LIN {X 0,Y 367.535,Z 523.641,A -85,B 0,C 180,E1 -12888.968,E2 -12888.968} C_VEL
LIN {X 0,Y 367.844,Z 521.457,A -85,B 0,C 180,E1 -12890.579,E2 -12890.579} C_VEL
LIN {X 0,Y 368.245,Z 517.815,A -85,B 0,C 180,E1 -12892.437,E2 -12892.437} C_VEL
LIN {X 0,Y 368.494,Z 515.813,A -85,B 0,C 180,E1 -12893.236,E2 -12893.236} C_VEL
LIN {X 0,Y 368.092,Z 513.552,A -85,B 0,C 180,E1 -12894.082,E2 -12894.082} C_VEL
LIN {X 0,Y 365.767,Z 509.524,A -85,B 0,C 180,E1 -12895.454,E2 -12895.454} C_VEL
LIN {X 0,Y 363.625,Z 504.962,A -85,B 0,C 180,E1 -12896.791,E2 -12896.791} C_VEL
LIN {X 0,Y 363.51,Z 501.685,A -85,B 0,C 180,E1 -12897.571,E2 -12897.571} C_VEL
LIN {X 0,Y 364.573,Z 493.787,A -85,B 0,C 180,E1 -12899.125,E2 -12899.125} C_VEL
LIN {X 0,Y 365.898,Z 483.754,A -85,B 0,C 180,E1 -12900.707,E2 -12900.707} C_VEL
LIN {X 0,Y 367.105,Z 474.13,A -85,B 0,C 180,E1 -12901.926,E2 -12901.926} C_VEL
LIN {X 0,Y 368.273,Z 463.742,A -85,B 0,C 180,E1 -12902.986,E2 -12902.986} C_VEL
LIN {X 0,Y 369.362,Z 451.282,A -85,B 0,C 180,E1 -12903.979,E2 -12903.979} C_VEL
LIN {X 0,Y 370.27,Z 438.997,A -85,B 0,C 180,E1 -12904.707,E2 -12904.707} C_VEL
LIN {X 0,Y 370.88,Z 426.339,A -85,B 0,C 180,E1 -12905.229,E2 -12905.229} C_VEL
LIN {X 0,Y 371.342,Z 411.465,A -85,B 0,C 180,E1 -12905.584,E2 -12905.584} C_VEL
LIN {X 0,Y 372.709,Z 340.608,A -85,B 0,C 180,E1 -12906.985,E2 -12906.985} C_VEL
LIN {X 0,Y 369.758,Z 328.428,A -85,B 0,C 180,E1 -12907.469,E2 -12907.469} C_VEL
LIN {X 0,Y 363.989,Z 314.826,A -85,B 0,C 180,E1 -12908.246,E2 -12908.246} C_VEL
LIN {X 0,Y 361.815,Z 305.413,A -85,B 0,C 180,E1 -12910.911,E2 -12910.911} C_VEL
LIN {X 0,Y 361.802,Z 305.418,A -85,B 0,C 180,E1 -12914.368,E2 -12914.368} C_VEL
LIN {X 0,Y 361.818,Z 305.416,A -85,B 0,C 180,E1 -12917.568,E2 -12917.568} C_VEL
LIN {X 0,Y 361.83,Z 305.417,A -85,B 0,C 180,E1 -12921.571,E2 -12921.571} C_VEL
LIN {X 0,Y 361.858,Z 305.393,A -85,B 0,C 180,E1 -12924.655,E2 -12924.655} C_VEL
LIN {X 0,Y 361.824,Z 305.409,A -85,B 0,C 180,E1 -12928.37,E2 -12928.37} C_VEL
LIN {X 0,Y 361.853,Z 305.409,A -85,B 0,C 180,E1 -12930.951,E2 -12930.951} C_VEL
LIN {X 0,Y 361.87,Z 305.403,A -85,B 0,C 180,E1 -12934.706,E2 -12934.706} C_VEL
LIN {X 0,Y 361.847,Z 305.405,A -85,B 0,C 180,E1 -12938.344,E2 -12938.344} C_VEL
LIN {X 0,Y 361.954,Z 305.397,A -85,B 0,C 180,E1 -12942.061,E2 -12942.061} C_VEL
LIN {X 0,Y 361.984,Z 305.396,A -85,B 0,C 180,E1 -12946.101,E2 -12946.101} C_VEL
LIN {X 0,Y 362.018,Z 305.389,A -85,B 0,C 180,E1 -12949.938,E2 -12949.938} C_VEL
LIN {X 0,Y 362.12,Z 305.366,A -85,B 0,C 180,E1 -12953.313,E2 -12953.313} C_VEL
LIN {X 0,Y 362.266,Z 305.351,A -85,B 0,C 180,E1 -12957.777,E2 -12957.777} C_VEL
LIN {X 0,Y 362.413,Z 305.337,A -85,B 0,C 180,E1 -12960,E2 -12960} C_VEL
LIN {X 0,Y 362.266,Z 305.355,A -85,B 0,C 180,E1 -12962.224,E2 -12962.224} C_VEL
LIN {X 0,Y 362.156,Z 305.371,A -85,B 0,C 180,E1 -12966.687,E2 -12966.687} C_VEL
LIN {X 0,Y 362.06,Z 305.376,A -85,B 0,C 180,E1 -12968.934,E2 -12968.934} C_VEL
LIN {X 0,Y 361.948,Z 305.397,A -85,B 0,C 180,E1 -12972.333,E2 -12972.333} C_VEL
LIN {X 0,Y 361.949,Z 305.39,A -85,B 0,C 180,E1 -12974.621,E2 -12974.621} C_VEL
LIN {X 0,Y 361.947,Z 305.392,A -85,B 0,C 180,E1 -12978.1,E2 -12978.1} C_VEL
LIN {X 0,Y 361.88,Z 305.405,A -85,B 0,C 180,E1 -12981.654,E2 -12981.654} C_VEL
LIN {X 0,Y 361.916,Z 305.404,A -85,B 0,C 180,E1 -12985.291,E2 -12985.291} C_VEL
LIN {X 0,Y 361.911,Z 305.394,A -85,B 0,C 180,E1 -12987.779,E2 -12987.779} C_VEL
LIN {X 0,Y 361.85,Z 305.405,A -85,B 0,C 180,E1 -12991.629,E2 -12991.629} C_VEL
LIN {X 0,Y 361.865,Z 305.408,A -85,B 0,C 180,E1 -12995.346,E2 -12995.346} C_VEL
LIN {X 0,Y 361.866,Z 305.409,A -85,B 0,C 180,E1 -12999.029,E2 -12999.029} C_VEL
LIN {X 0,Y 361.849,Z 305.408,A -85,B 0,C 180,E1 -13002.437,E2 -13002.437} C_VEL
LIN {X 0,Y 361.891,Z 305.393,A -85,B 0,C 180,E1 -13005.935,E2 -13005.935} C_VEL
LIN {X 0,Y 361.899,Z 305.401,A -85,B 0,C 180,E1 -13009.233,E2 -13009.233} C_VEL
LIN {X 0,Y 361.863,Z 305.407,A -85,B 0,C 180,E1 -13012.984,E2 -13012.984} C_VEL
LIN {X 0,Y 361.853,Z 305.407,A -85,B 0,C 180,E1 -13016.633,E2 -13016.633} C_VEL
LIN {X 0,Y 361.904,Z 305.519,A -85,B 0,C 180,E1 -13018.541,E2 -13018.541} C_VEL
LIN {X 0,Y 364.797,Z 317.675,A -85,B 0,C 180,E1 -13021.838,E2 -13021.838} C_VEL
LIN {X 0,Y 366.633,Z 327.228,A -85,B 0,C 180,E1 -13024.283,E2 -13024.283} C_VEL
LIN {X 0,Y 366.075,Z 334.395,A -85,B 0,C 180,E1 -13025.925,E2 -13025.925} C_VEL
LIN {X 0,Y 365.502,Z 339.003,A -85,B 0,C 180,E1 -13026.956,E2 -13026.956} C_VEL
LIN {X 0,Y 369.726,Z 359.775,A -85,B 0,C 180,E1 -13027.733,E2 -13027.733} C_VEL
LIN {X 0,Y 372.145,Z 375.173,A -85,B 0,C 180,E1 -13028.239,E2 -13028.239} C_VEL
LIN {X 0,Y 370.626,Z 447.548,A -85,B 0,C 180,E1 -13029.683,E2 -13029.683} C_VEL
LIN {X 0,Y 369.963,Z 460.734,A -85,B 0,C 180,E1 -13030.152,E2 -13030.152} C_VEL
LIN {X 0,Y 368.926,Z 473.426,A -85,B 0,C 180,E1 -13030.817,E2 -13030.817} C_VEL
LIN {X 0,Y 367.825,Z 484.734,A -85,B 0,C 180,E1 -13031.625,E2 -13031.625} C_VEL
LIN {X 0,Y 366.507,Z 496.397,A -85,B 0,C 180,E1 -13032.711,E2 -13032.711} C_VEL
LIN {X 0,Y 365.178,Z 506.891,A -85,B 0,C 180,E1 -13033.941,E2 -13033.941} C_VEL
LIN {X 0,Y 364.137,Z 515.532,A -85,B 0,C 180,E1 -13035.191,E2 -13035.191} C_VEL
LIN {X 0,Y 363.149,Z 523.447,A -85,B 0,C 180,E1 -13036.573,E2 -13036.573} C_VEL
LIN {X 0,Y 362.018,Z 531.267,A -85,B 0,C 180,E1 -13038.24,E2 -13038.24} C_VEL
LIN {X 0,Y 361.281,Z 537.541,A -85,B 0,C 180,E1 -13039.919,E2 -13039.919} C_VEL
LIN {X 0,Y 360.808,Z 542.555,A -85,B 0,C 180,E1 -13041.601,E2 -13041.601} C_VEL
LIN {X 0,Y 360.498,Z 546.453,A -85,B 0,C 180,E1 -13043.284,E2 -13043.284} C_VEL
LIN {X 0,Y 360.365,Z 550.078,A -85,B 0,C 180,E1 -13045.528,E2 -13045.528} C_VEL
LIN {X 0,Y 360.301,Z 551.276,A -85,B 0,C 180,E1 -13046.647,E2 -13046.647} C_VEL
LIN {X 0,Y 360.358,Z 552.408,A -85,B 0,C 180,E1 -13048.884,E2 -13048.884} C_VEL
LIN {X 0,Y 360.423,Z 552.394,A -85,B 0,C 180,E1 -13050.002,E2 -13050.002} C_VEL
LIN {X 0,Y 360.39,Z 551.986,A -85,B 0,C 180,E1 -13051.119,E2 -13051.119} C_VEL
LIN {X 0,Y 360.327,Z 551.136,A -85,B 0,C 180,E1 -13052.237,E2 -13052.237} C_VEL
LIN {X 0,Y 360.322,Z 549.88,A -85,B 0,C 180,E1 -13053.356,E2 -13053.356} C_VEL
LIN {X 0,Y 360.376,Z 547.203,A -85,B 0,C 180,E1 -13055.036,E2 -13055.036} C_VEL
LIN {X 0,Y 360.499,Z 543.49,A -85,B 0,C 180,E1 -13056.719,E2 -13056.719} C_VEL
LIN {X 0,Y 360.749,Z 538.639,A -85,B 0,C 180,E1 -13058.403,E2 -13058.403} C_VEL
LIN {X 0,Y 361.16,Z 532.502,A -85,B 0,C 180,E1 -13060.088,E2 -13060.088} C_VEL
LIN {X 0,Y 361.765,Z 524.858,A -85,B 0,C 180,E1 -13061.772,E2 -13061.772} C_VEL
LIN {X 0,Y 362.468,Z 517.035,A -85,B 0,C 180,E1 -13063.171,E2 -13063.171} C_VEL
LIN {X 0,Y 363.412,Z 507.472,A -85,B 0,C 180,E1 -13064.562,E2 -13064.562} C_VEL
LIN {X 0,Y 364.246,Z 496.828,A -85,B 0,C 180,E1 -13065.817,E2 -13065.817} C_VEL
LIN {X 0,Y 365.222,Z 484.96,A -85,B 0,C 180,E1 -13066.922,E2 -13066.922} C_VEL
LIN {X 0,Y 366.15,Z 472.226,A -85,B 0,C 180,E1 -13067.814,E2 -13067.814} C_VEL
LIN {X 0,Y 366.97,Z 459.529,A -85,B 0,C 180,E1 -13068.459,E2 -13068.459} C_VEL
LIN {X 0,Y 367.431,Z 447.489,A -85,B 0,C 180,E1 -13068.868,E2 -13068.868} C_VEL
LIN {X 0,Y 368.577,Z 374.068,A -85,B 0,C 180,E1 -13070.315,E2 -13070.315} C_VEL
LIN {X 0,Y 363.856,Z 339.626,A -85,B 0,C 180,E1 -13071.264,E2 -13071.264} C_VEL
LIN {X 0,Y 365.182,Z 323.829,A -85,B 0,C 180,E1 -13074.747,E2 -13074.747} C_VEL
LIN {X 0,Y 364.808,Z 319.729,A -85,B 0,C 180,E1 -13075.697,E2 -13075.697} C_VEL
LIN {X 0,Y 362.061,Z 305.992,A -85,B 0,C 180,E1 -13079.032,E2 -13079.032} C_VEL
LIN {X 0,Y 361.931,Z 305.4,A -85,B 0,C 180,E1 -13079.222,E2 -13079.222} C_VEL
LIN {X 0,Y 361.865,Z 305.405,A -85,B 0,C 180,E1 -13083.37,E2 -13083.37} C_VEL
LIN {X 0,Y 361.872,Z 305.405,A -85,B 0,C 180,E1 -13087.019,E2 -13087.019} C_VEL
LIN {X 0,Y 361.86,Z 305.407,A -85,B 0,C 180,E1 -13089.862,E2 -13089.862} C_VEL
LIN {X 0,Y 361.842,Z 305.412,A -85,B 0,C 180,E1 -13092.83,E2 -13092.83} C_VEL
LIN {X 0,Y 361.824,Z 305.411,A -85,B 0,C 180,E1 -13095.947,E2 -13095.947} C_VEL
LIN {X 0,Y 361.842,Z 305.41,A -85,B 0,C 180,E1 -13099.245,E2 -13099.245} C_VEL
LIN {X 0,Y 361.87,Z 305.411,A -85,B 0,C 180,E1 -13102.778,E2 -13102.778} C_VEL
LIN {X 0,Y 361.86,Z 305.406,A -85,B 0,C 180,E1 -13105.72,E2 -13105.72} C_VEL
LIN {X 0,Y 361.881,Z 305.405,A -85,B 0,C 180,E1 -13109.672,E2 -13109.672} C_VEL
LIN {X 0,Y 361.961,Z 305.398,A -85,B 0,C 180,E1 -13113.475,E2 -13113.475} C_VEL
LIN {X 0,Y 361.886,Z 305.407,A -85,B 0,C 180,E1 -13117.144,E2 -13117.144} C_VEL
LIN {X 0,Y 361.892,Z 305.402,A -85,B 0,C 180,E1 -13120.722,E2 -13120.722} C_VEL
LIN {X 0,Y 361.95,Z 305.396,A -85,B 0,C 180,E1 -13124.226,E2 -13124.226} C_VEL
LIN {X 0,Y 362.006,Z 305.388,A -85,B 0,C 180,E1 -13126.528,E2 -13126.528} C_VEL
LIN {X 0,Y 362.036,Z 305.389,A -85,B 0,C 180,E1 -13129.938,E2 -13129.938} C_VEL
LIN {X 0,Y 362.131,Z 305.373,A -85,B 0,C 180,E1 -13133.313,E2 -13133.313} C_VEL
LIN {X 0,Y 362.286,Z 305.357,A -85,B 0,C 180,E1 -13137.776,E2 -13137.776} C_VEL
LIN {X 0,Y 362.43,Z 305.341,A -85,B 0,C 180,E1 -13140,E2 -13140} C_VEL
LIN {X 0,Y 362.285,Z 305.36,A -85,B 0,C 180,E1 -13142.223,E2 -13142.223} C_VEL
LIN {X 0,Y 362.154,Z 305.372,A -85,B 0,C 180,E1 -13146.686,E2 -13146.686} C_VEL
LIN {X 0,Y 362.006,Z 305.391,A -85,B 0,C 180,E1 -13150.063,E2 -13150.063} C_VEL
LIN {X 0,Y 362.004,Z 305.389,A -85,B 0,C 180,E1 -13153.898,E2 -13153.898} C_VEL
LIN {X 0,Y 361.934,Z 305.401,A -85,B 0,C 180,E1 -13156.934,E2 -13156.934} C_VEL
LIN {X 0,Y 361.892,Z 305.405,A -85,B 0,C 180,E1 -13160.46,E2 -13160.46} C_VEL
LIN {X 0,Y 361.899,Z 305.401,A -85,B 0,C 180,E1 -13164.112,E2 -13164.112} C_VEL
LIN {X 0,Y 361.947,Z 305.399,A -85,B 0,C 180,E1 -13166.721,E2 -13166.721} C_VEL
LIN {X 0,Y 361.878,Z 305.404,A -85,B 0,C 180,E1 -13170.327,E2 -13170.327} C_VEL
LIN {X 0,Y 361.859,Z 305.406,A -85,B 0,C 180,E1 -13174.28,E2 -13174.28} C_VEL
LIN {X 0,Y 361.868,Z 305.411,A -85,B 0,C 180,E1 -13177.222,E2 -13177.222} C_VEL
LIN {X 0,Y 361.84,Z 305.409,A -85,B 0,C 180,E1 -13180.755,E2 -13180.755} C_VEL
LIN {X 0,Y 361.821,Z 305.411,A -85,B 0,C 180,E1 -13184.368,E2 -13184.368} C_VEL
LIN {X 0,Y 361.84,Z 305.414,A -85,B 0,C 180,E1 -13187.567,E2 -13187.567} C_VEL
LIN {X 0,Y 361.872,Z 305.405,A -85,B 0,C 180,E1 -13190.973,E2 -13190.973} C_VEL
LIN {X 0,Y 361.878,Z 305.404,A -85,B 0,C 180,E1 -13194.654,E2 -13194.654} C_VEL
LIN {X 0,Y 361.842,Z 305.411,A -85,B 0,C 180,E1 -13198.369,E2 -13198.369} C_VEL
LIN {X 0,Y 361.912,Z 305.406,A -85,B 0,C 180,E1 -13202.22,E2 -13202.22} C_VEL
LIN {X 0,Y 361.931,Z 305.399,A -85,B 0,C 180,E1 -13204.709,E2 -13204.709} C_VEL
LIN {X 0,Y 361.902,Z 305.408,A -85,B 0,C 180,E1 -13208.346,E2 -13208.346} C_VEL
LIN {X 0,Y 361.971,Z 305.395,A -85,B 0,C 180,E1 -13212.06,E2 -13212.06} C_VEL
LIN {X 0,Y 362,Z 305.39,A -85,B 0,C 180,E1 -13216.1,E2 -13216.1} C_VEL
LIN {X 0,Y 362.002,Z 305.389,A -85,B 0,C 180,E1 -13219.936,E2 -13219.936} C_VEL
LIN {X 0,Y 362.087,Z 305.512,A -85,B 0,C 180,E1 -13221.461,E2 -13221.461} C_VEL
LIN {X 0,Y 363.79,Z 314.739,A -85,B 0,C 180,E1 -13223.84,E2 -13223.84} C_VEL
LIN {X 0,Y 365.852,Z 322.952,A -85,B 0,C 180,E1 -13224.111,E2 -13224.111} C_VEL
LIN {X 0,Y 369.039,Z 340.026,A -85,B 0,C 180,E1 -13224.613,E2 -13224.613} C_VEL
LIN {X 0,Y 367.633,Z 422.051,A -85,B 0,C 180,E1 -13226.231,E2 -13226.231} C_VEL
LIN {X 0,Y 367.087,Z 435.227,A -85,B 0,C 180,E1 -13226.706,E2 -13226.706} C_VEL
LIN {X 0,Y 366.558,Z 447.799,A -85,B 0,C 180,E1 -13227.388,E2 -13227.388} C_VEL
LIN {X 0,Y 365.821,Z 459.62,A -85,B 0,C 180,E1 -13228.258,E2 -13228.258} C_VEL
LIN {X 0,Y 364.903,Z 470.713,A -85,B 0,C 180,E1 -13229.309,E2 -13229.309} C_VEL
LIN {X 0,Y 363.959,Z 481.189,A -85,B 0,C 180,E1 -13230.552,E2 -13230.552} C_VEL
LIN {X 0,Y 363.107,Z 490.613,A -85,B 0,C 180,E1 -13231.939,E2 -13231.939} C_VEL
LIN {X 0,Y 362.216,Z 499.705,A -85,B 0,C 180,E1 -13233.614,E2 -13233.614} C_VEL
LIN {X 0,Y 361.528,Z 507.037,A -85,B 0,C 180,E1 -13235.296,E2 -13235.296} C_VEL
LIN {X 0,Y 361.166,Z 513.125,A -85,B 0,C 180,E1 -13237.061,E2 -13237.061} C_VEL
LIN {X 0,Y 360.72,Z 518.155,A -85,B 0,C 180,E1 -13238.965,E2 -13238.965} C_VEL
LIN {X 0,Y 360.511,Z 520.505,A -85,B 0,C 180,E1 -13240.103,E2 -13240.103} C_VEL
LIN {X 0,Y 360.403,Z 522.413,A -85,B 0,C 180,E1 -13241.243,E2 -13241.243} C_VEL
LIN {X 0,Y 360.295,Z 524.217,A -85,B 0,C 180,E1 -13242.758,E2 -13242.758} C_VEL
LIN {X 0,Y 360.201,Z 525.48,A -85,B 0,C 180,E1 -13244.692,E2 -13244.692} C_VEL
LIN {X 0,Y 360.218,Z 525.667,A -85,B 0,C 180,E1 -13245.85,E2 -13245.85} C_VEL
LIN {X 0,Y 360.27,Z 525.382,A -85,B 0,C 180,E1 -13247.085,E2 -13247.085} C_VEL
LIN {X 0,Y 360.499,Z 523.665,A -85,B 0,C 180,E1 -13249.353,E2 -13249.353} C_VEL
LIN {X 0,Y 360.805,Z 521.693,A -85,B 0,C 180,E1 -13250.776,E2 -13250.776} C_VEL
LIN {X 0,Y 361.311,Z 517.534,A -85,B 0,C 180,E1 -13252.892,E2 -13252.892} C_VEL
LIN {X 0,Y 361.97,Z 512.677,A -85,B 0,C 180,E1 -13254.671,E2 -13254.671} C_VEL
LIN {X 0,Y 362.839,Z 506.421,A -85,B 0,C 180,E1 -13256.453,E2 -13256.453} C_VEL
LIN {X 0,Y 363.51,Z 501.685,A -85,B 0,C 180,E1 -13257.571,E2 -13257.571} C_VEL
LIN {X 0,Y 363.434,Z 498.283,A -85,B 0,C 180,E1 -13258.333,E2 -13258.333} C_VEL
LIN {X 0,Y 361.524,Z 492.515,A -85,B 0,C 180,E1 -13259.574,E2 -13259.574} C_VEL
LIN {X 0,Y 359.6,Z 486.162,A -85,B 0,C 180,E1 -13260.746,E2 -13260.746} C_VEL
LIN {X 0,Y 359.49,Z 481.841,A -85,B 0,C 180,E1 -13261.388,E2 -13261.388} C_VEL
LIN {X 0,Y 360.854,Z 470.901,A -85,B 0,C 180,E1 -13262.712,E2 -13262.712} C_VEL
LIN {X 0,Y 362.095,Z 459.975,A -85,B 0,C 180,E1 -13263.76,E2 -13263.76} C_VEL
LIN {X 0,Y 363.096,Z 448.05,A -85,B 0,C 180,E1 -13264.648,E2 -13264.648} C_VEL
LIN {X 0,Y 363.996,Z 435.03,A -85,B 0,C 180,E1 -13265.352,E2 -13265.352} C_VEL
LIN {X 0,Y 364.566,Z 422.079,A -85,B 0,C 180,E1 -13265.82,E2 -13265.82} C_VEL
LIN {X 0,Y 366.353,Z 341.95,A -85,B 0,C 180,E1 -13267.441,E2 -13267.441} C_VEL
LIN {X 0,Y 363.742,Z 331.236,A -85,B 0,C 180,E1 -13267.882,E2 -13267.882} C_VEL
LIN {X 0,Y 356.868,Z 315.147,A -85,B 0,C 180,E1 -13268.828,E2 -13268.828} C_VEL
LIN {X 0,Y 354.764,Z 306.292,A -85,B 0,C 180,E1 -13271.421,E2 -13271.421} C_VEL
LIN {X 0,Y 354.749,Z 306.296,A -85,B 0,C 180,E1 -13274.504,E2 -13274.504} C_VEL
LIN {X 0,Y 354.776,Z 306.295,A -85,B 0,C 180,E1 -13277.66,E2 -13277.66} C_VEL
LIN {X 0,Y 354.773,Z 306.293,A -85,B 0,C 180,E1 -13280.661,E2 -13280.661} C_VEL
LIN {X 0,Y 354.806,Z 306.271,A -85,B 0,C 180,E1 -13284.301,E2 -13284.301} C_VEL
LIN {X 0,Y 354.774,Z 306.294,A -85,B 0,C 180,E1 -13287.666,E2 -13287.666} C_VEL
LIN {X 0,Y 354.788,Z 306.288,A -85,B 0,C 180,E1 -13291.614,E2 -13291.614} C_VEL
LIN {X 0,Y 354.821,Z 306.281,A -85,B 0,C 180,E1 -13295.656,E2 -13295.656} C_VEL
LIN {X 0,Y 354.813,Z 306.279,A -85,B 0,C 180,E1 -13299.113,E2 -13299.113} C_VEL
LIN {X 0,Y 354.884,Z 306.271,A -85,B 0,C 180,E1 -13302.719,E2 -13302.719} C_VEL
LIN {X 0,Y 354.937,Z 306.272,A -85,B 0,C 180,E1 -13306.255,E2 -13306.255} C_VEL
LIN {X 0,Y 354.965,Z 306.266,A -85,B 0,C 180,E1 -13309.736,E2 -13309.736} C_VEL
LIN {X 0,Y 355.085,Z 306.242,A -85,B 0,C 180,E1 -13313.18,E2 -13313.18} C_VEL
LIN {X 0,Y 355.229,Z 306.227,A -85,B 0,C 180,E1 -13317.733,E2 -13317.733} C_VEL
LIN {X 0,Y 355.383,Z 306.212,A -85,B 0,C 180,E1 -13320,E2 -13320} C_VEL
LIN {X 0,Y 355.229,Z 306.23,A -85,B 0,C 180,E1 -13322.268,E2 -13322.268} C_VEL
LIN {X 0,Y 355.123,Z 306.246,A -85,B 0,C 180,E1 -13326.82,E2 -13326.82} C_VEL
LIN {X 0,Y 355.002,Z 306.255,A -85,B 0,C 180,E1 -13329.113,E2 -13329.113} C_VEL
LIN {X 0,Y 354.908,Z 306.271,A -85,B 0,C 180,E1 -13332.582,E2 -13332.582} C_VEL
LIN {X 0,Y 354.876,Z 306.278,A -85,B 0,C 180,E1 -13336.097,E2 -13336.097} C_VEL
LIN {X 0,Y 354.894,Z 306.27,A -85,B 0,C 180,E1 -13338.473,E2 -13338.473} C_VEL
LIN {X 0,Y 354.822,Z 306.284,A -85,B 0,C 180,E1 -13342.107,E2 -13342.107} C_VEL
LIN {X 0,Y 354.888,Z 306.277,A -85,B 0,C 180,E1 -13345.829,E2 -13345.829} C_VEL
LIN {X 0,Y 354.844,Z 306.285,A -85,B 0,C 180,E1 -13349.68,E2 -13349.68} C_VEL
LIN {X 0,Y 354.82,Z 306.29,A -85,B 0,C 180,E1 -13353.684,E2 -13353.684} C_VEL
LIN {X 0,Y 354.792,Z 306.288,A -85,B 0,C 180,E1 -13356.461,E2 -13356.461} C_VEL
LIN {X 0,Y 354.815,Z 306.287,A -85,B 0,C 180,E1 -13359.425,E2 -13359.425} C_VEL
LIN {X 0,Y 354.8,Z 306.287,A -85,B 0,C 180,E1 -13362.872,E2 -13362.872} C_VEL
LIN {X 0,Y 354.833,Z 306.272,A -85,B 0,C 180,E1 -13366.117,E2 -13366.117} C_VEL
LIN {X 0,Y 354.851,Z 306.279,A -85,B 0,C 180,E1 -13369.191,E2 -13369.191} C_VEL
LIN {X 0,Y 354.803,Z 306.29,A -85,B 0,C 180,E1 -13372.404,E2 -13372.404} C_VEL
LIN {X 0,Y 354.807,Z 306.292,A -85,B 0,C 180,E1 -13374.943,E2 -13374.943} C_VEL
LIN {X 0,Y 354.862,Z 306.413,A -85,B 0,C 180,E1 -13378.037,E2 -13378.037} C_VEL
LIN {X 0,Y 357.895,Z 319.073,A -85,B 0,C 180,E1 -13381.565,E2 -13381.565} C_VEL
LIN {X 0,Y 359.716,Z 328.332,A -85,B 0,C 180,E1 -13383.993,E2 -13383.993} C_VEL
LIN {X 0,Y 359.647,Z 331.913,A -85,B 0,C 180,E1 -13384.85,E2 -13384.85} C_VEL
LIN {X 0,Y 358.826,Z 338.677,A -85,B 0,C 180,E1 -13386.402,E2 -13386.402} C_VEL
LIN {X 0,Y 363.247,Z 360.149,A -85,B 0,C 180,E1 -13387.246,E2 -13387.246} C_VEL
LIN {X 0,Y 365.738,Z 376.161,A -85,B 0,C 180,E1 -13387.786,E2 -13387.786} C_VEL
LIN {X 0,Y 364.147,Z 447.404,A -85,B 0,C 180,E1 -13389.231,E2 -13389.231} C_VEL
LIN {X 0,Y 363.443,Z 460.548,A -85,B 0,C 180,E1 -13389.706,E2 -13389.706} C_VEL
LIN {X 0,Y 362.33,Z 473.223,A -85,B 0,C 180,E1 -13390.381,E2 -13390.381} C_VEL
LIN {X 0,Y 361.128,Z 485.309,A -85,B 0,C 180,E1 -13391.272,E2 -13391.272} C_VEL
LIN {X 0,Y 359.74,Z 496.806,A -85,B 0,C 180,E1 -13392.375,E2 -13392.375} C_VEL
LIN {X 0,Y 358.362,Z 507.184,A -85,B 0,C 180,E1 -13393.627,E2 -13393.627} C_VEL
LIN {X 0,Y 357.23,Z 516.028,A -85,B 0,C 180,E1 -13394.948,E2 -13394.948} C_VEL
LIN {X 0,Y 356.027,Z 524.943,A -85,B 0,C 180,E1 -13396.59,E2 -13396.59} C_VEL
LIN {X 0,Y 354.887,Z 532.393,A -85,B 0,C 180,E1 -13398.29,E2 -13398.29} C_VEL
LIN {X 0,Y 354.067,Z 539.302,A -85,B 0,C 180,E1 -13400.288,E2 -13400.288} C_VEL
LIN {X 0,Y 353.622,Z 543.886,A -85,B 0,C 180,E1 -13402.005,E2 -13402.005} C_VEL
LIN {X 0,Y 353.324,Z 547.878,A -85,B 0,C 180,E1 -13404.021,E2 -13404.021} C_VEL
LIN {X 0,Y 353.278,Z 549.899,A -85,B 0,C 180,E1 -13405.438,E2 -13405.438} C_VEL
LIN {X 0,Y 353.223,Z 551.062,A -85,B 0,C 180,E1 -13406.58,E2 -13406.58} C_VEL
LIN {X 0,Y 353.26,Z 552.152,A -85,B 0,C 180,E1 -13408.862,E2 -13408.862} C_VEL
LIN {X 0,Y 353.328,Z 552.119,A -85,B 0,C 180,E1 -13410.002,E2 -13410.002} C_VEL
LIN {X 0,Y 353.292,Z 551.68,A -85,B 0,C 180,E1 -13411.142,E2 -13411.142} C_VEL
LIN {X 0,Y 353.244,Z 549.527,A -85,B 0,C 180,E1 -13413.423,E2 -13413.423} C_VEL
LIN {X 0,Y 353.28,Z 546.808,A -85,B 0,C 180,E1 -13415.138,E2 -13415.138} C_VEL
LIN {X 0,Y 353.418,Z 543.05,A -85,B 0,C 180,E1 -13416.854,E2 -13416.854} C_VEL
LIN {X 0,Y 353.686,Z 538.151,A -85,B 0,C 180,E1 -13418.572,E2 -13418.572} C_VEL
LIN {X 0,Y 354.125,Z 531.962,A -85,B 0,C 180,E1 -13420.291,E2 -13420.291} C_VEL
LIN {X 0,Y 354.776,Z 524.252,A -85,B 0,C 180,E1 -13422.007,E2 -13422.007} C_VEL
LIN {X 0,Y 355.506,Z 516.342,A -85,B 0,C 180,E1 -13423.433,E2 -13423.433} C_VEL
LIN {X 0,Y 356.461,Z 506.675,A -85,B 0,C 180,E1 -13424.853,E2 -13424.853} C_VEL
LIN {X 0,Y 357.347,Z 495.923,A -85,B 0,C 180,E1 -13426.13,E2 -13426.13} C_VEL
LIN {X 0,Y 358.244,Z 485.538,A -85,B 0,C 180,E1 -13427.115,E2 -13427.115} C_VEL
LIN {X 0,Y 359.198,Z 473.124,A -85,B 0,C 180,E1 -13428.024,E2 -13428.024} C_VEL
LIN {X 0,Y 360.083,Z 460.064,A -85,B 0,C 180,E1 -13428.714,E2 -13428.714} C_VEL
LIN {X 0,Y 360.602,Z 447.283,A -85,B 0,C 180,E1 -13429.166,E2 -13429.166} C_VEL
LIN {X 0,Y 361.742,Z 374.325,A -85,B 0,C 180,E1 -13430.631,E2 -13430.631} C_VEL
LIN {X 0,Y 356.926,Z 339.462,A -85,B 0,C 180,E1 -13431.596,E2 -13431.596} C_VEL
LIN {X 0,Y 358.216,Z 324.541,A -85,B 0,C 180,E1 -13434.951,E2 -13434.951} C_VEL
LIN {X 0,Y 357.483,Z 319.09,A -85,B 0,C 180,E1 -13436.255,E2 -13436.255} C_VEL
LIN {X 0,Y 354.891,Z 306.277,A -85,B 0,C 180,E1 -13439.474,E2 -13439.474} C_VEL
LIN {X 0,Y 354.812,Z 306.285,A -85,B 0,C 180,E1 -13443.703,E2 -13443.703} C_VEL
LIN {X 0,Y 354.804,Z 306.291,A -85,B 0,C 180,E1 -13446.46,E2 -13446.46} C_VEL
LIN {X 0,Y 354.831,Z 306.282,A -85,B 0,C 180,E1 -13449.424,E2 -13449.424} C_VEL
LIN {X 0,Y 354.794,Z 306.29,A -85,B 0,C 180,E1 -13452.868,E2 -13452.868} C_VEL
LIN {X 0,Y 354.773,Z 306.29,A -85,B 0,C 180,E1 -13456.104,E2 -13456.104} C_VEL
LIN {X 0,Y 354.795,Z 306.289,A -85,B 0,C 180,E1 -13459.18,E2 -13459.18} C_VEL
LIN {X 0,Y 354.813,Z 306.286,A -85,B 0,C 180,E1 -13462.403,E2 -13462.403} C_VEL
LIN {X 0,Y 354.818,Z 306.29,A -85,B 0,C 180,E1 -13464.941,E2 -13464.941} C_VEL
LIN {X 0,Y 354.799,Z 306.286,A -85,B 0,C 180,E1 -13468.406,E2 -13468.406} C_VEL
LIN {X 0,Y 354.856,Z 306.281,A -85,B 0,C 180,E1 -13471.619,E2 -13471.619} C_VEL
LIN {X 0,Y 354.905,Z 306.272,A -85,B 0,C 180,E1 -13474.173,E2 -13474.173} C_VEL
LIN {X 0,Y 354.823,Z 306.284,A -85,B 0,C 180,E1 -13477.893,E2 -13477.893} C_VEL
LIN {X 0,Y 354.897,Z 306.276,A -85,B 0,C 180,E1 -13481.908,E2 -13481.908} C_VEL
LIN {X 0,Y 354.95,Z 306.27,A -85,B 0,C 180,E1 -13485.981,E2 -13485.981} C_VEL
LIN {X 0,Y 354.983,Z 306.269,A -85,B 0,C 180,E1 -13489.736,E2 -13489.736} C_VEL
LIN {X 0,Y 355.096,Z 306.249,A -85,B 0,C 180,E1 -13493.18,E2 -13493.18} C_VEL
LIN {X 0,Y 355.249,Z 306.233,A -85,B 0,C 180,E1 -13497.732,E2 -13497.732} C_VEL
LIN {X 0,Y 355.379,Z 306.219,A -85,B 0,C 180,E1 -13500,E2 -13500} C_VEL
LIN {X 0,Y 355.248,Z 306.236,A -85,B 0,C 180,E1 -13502.267,E2 -13502.267} C_VEL
LIN {X 0,Y 355.117,Z 306.248,A -85,B 0,C 180,E1 -13506.819,E2 -13506.819} C_VEL
LIN {X 0,Y 354.962,Z 306.27,A -85,B 0,C 180,E1 -13510.264,E2 -13510.264} C_VEL
LIN {X 0,Y 354.949,Z 306.268,A -85,B 0,C 180,E1 -13514.018,E2 -13514.018} C_VEL
LIN {X 0,Y 354.896,Z 306.275,A -85,B 0,C 180,E1 -13518.092,E2 -13518.092} C_VEL
LIN {X 0,Y 354.823,Z 306.283,A -85,B 0,C 180,E1 -13522.107,E2 -13522.107} C_VEL
LIN {X 0,Y 354.904,Z 306.273,A -85,B 0,C 180,E1 -13525.827,E2 -13525.827} C_VEL
LIN {X 0,Y 354.823,Z 306.284,A -85,B 0,C 180,E1 -13529.681,E2 -13529.681} C_VEL
LIN {X 0,Y 354.811,Z 306.286,A -85,B 0,C 180,E1 -13533.701,E2 -13533.701} C_VEL
LIN {X 0,Y 354.802,Z 306.285,A -85,B 0,C 180,E1 -13536.459,E2 -13536.459} C_VEL
LIN {X 0,Y 354.829,Z 306.289,A -85,B 0,C 180,E1 -13539.423,E2 -13539.423} C_VEL
LIN {X 0,Y 354.793,Z 306.287,A -85,B 0,C 180,E1 -13542.866,E2 -13542.866} C_VEL
LIN {X 0,Y 354.771,Z 306.291,A -85,B 0,C 180,E1 -13546.103,E2 -13546.103} C_VEL
LIN {X 0,Y 354.792,Z 306.288,A -85,B 0,C 180,E1 -13549.178,E2 -13549.178} C_VEL
LIN {X 0,Y 354.81,Z 306.285,A -85,B 0,C 180,E1 -13552.402,E2 -13552.402} C_VEL
LIN {X 0,Y 354.816,Z 306.283,A -85,B 0,C 180,E1 -13554.94,E2 -13554.94} C_VEL
LIN {X 0,Y 354.797,Z 306.289,A -85,B 0,C 180,E1 -13558.404,E2 -13558.404} C_VEL
LIN {X 0,Y 354.85,Z 306.281,A -85,B 0,C 180,E1 -13561.617,E2 -13561.617} C_VEL
LIN {X 0,Y 354.902,Z 306.279,A -85,B 0,C 180,E1 -13564.171,E2 -13564.171} C_VEL
LIN {X 0,Y 354.842,Z 306.282,A -85,B 0,C 180,E1 -13567.893,E2 -13567.893} C_VEL
LIN {X 0,Y 354.926,Z 306.271,A -85,B 0,C 180,E1 -13571.89,E2 -13571.89} C_VEL
LIN {X 0,Y 354.945,Z 306.268,A -85,B 0,C 180,E1 -13575.98,E2 -13575.98} C_VEL
LIN {X 0,Y 354.958,Z 306.266,A -85,B 0,C 180,E1 -13579.734,E2 -13579.734} C_VEL
LIN {X 0,Y 355.039,Z 306.372,A -85,B 0,C 180,E1 -13581.214,E2 -13581.214} C_VEL
LIN {X 0,Y 356.619,Z 314.782,A -85,B 0,C 180,E1 -13583.463,E2 -13583.463} C_VEL
LIN {X 0,Y 359.064,Z 323.796,A -85,B 0,C 180,E1 -13583.786,E2 -13583.786} C_VEL
LIN {X 0,Y 362.265,Z 340.51,A -85,B 0,C 180,E1 -13584.294,E2 -13584.294} C_VEL
LIN {X 0,Y 360.778,Z 422.793,A -85,B 0,C 180,E1 -13585.949,E2 -13585.949} C_VEL
LIN {X 0,Y 360.236,Z 435.8,A -85,B 0,C 180,E1 -13586.433,E2 -13586.433} C_VEL
LIN {X 0,Y 359.676,Z 448.304,A -85,B 0,C 180,E1 -13587.128,E2 -13587.128} C_VEL
LIN {X 0,Y 358.927,Z 460.083,A -85,B 0,C 180,E1 -13588.017,E2 -13588.017} C_VEL
LIN {X 0,Y 357.923,Z 471.766,A -85,B 0,C 180,E1 -13589.155,E2 -13589.155} C_VEL
LIN {X 0,Y 356.945,Z 482.114,A -85,B 0,C 180,E1 -13590.421,E2 -13590.421} C_VEL
LIN {X 0,Y 356.137,Z 490.558,A -85,B 0,C 180,E1 -13591.695,E2 -13591.695} C_VEL
LIN {X 0,Y 355.203,Z 499.714,A -85,B 0,C 180,E1 -13593.401,E2 -13593.401} C_VEL
LIN {X 0,Y 354.509,Z 507.086,A -85,B 0,C 180,E1 -13595.116,E2 -13595.116} C_VEL
LIN {X 0,Y 354.086,Z 513.653,A -85,B 0,C 180,E1 -13597.063,E2 -13597.063} C_VEL
LIN {X 0,Y 353.598,Z 518.931,A -85,B 0,C 180,E1 -13599.147,E2 -13599.147} C_VEL
LIN {X 0,Y 353.387,Z 521.21,A -85,B 0,C 180,E1 -13600.309,E2 -13600.309} C_VEL
LIN {X 0,Y 353.296,Z 522.989,A -85,B 0,C 180,E1 -13601.472,E2 -13601.472} C_VEL
LIN {X 0,Y 353.198,Z 524.537,A -85,B 0,C 180,E1 -13602.836,E2 -13602.836} C_VEL
LIN {X 0,Y 353.098,Z 525.823,A -85,B 0,C 180,E1 -13604.994,E2 -13604.994} C_VEL
LIN {X 0,Y 353.181,Z 525.637,A -85,B 0,C 180,E1 -13607.224,E2 -13607.224} C_VEL
LIN {X 0,Y 353.301,Z 524.847,A -85,B 0,C 180,E1 -13608.557,E2 -13608.557} C_VEL
LIN {X 0,Y 353.504,Z 523.632,A -85,B 0,C 180,E1 -13609.752,E2 -13609.752} C_VEL
LIN {X 0,Y 353.878,Z 520.976,A -85,B 0,C 180,E1 -13611.553,E2 -13611.553} C_VEL
LIN {X 0,Y 354.406,Z 517.2,A -85,B 0,C 180,E1 -13613.364,E2 -13613.364} C_VEL
LIN {X 0,Y 355.13,Z 512.181,A -85,B 0,C 180,E1 -13615.179,E2 -13615.179} C_VEL
LIN {X 0,Y 356.047,Z 505.745,A -85,B 0,C 180,E1 -13616.998,E2 -13616.998} C_VEL
LIN {X 0,Y 357.095,Z 499.084,A -85,B 0,C 180,E1 -13618.505,E2 -13618.505} C_VEL
LIN {X 0,Y 358.199,Z 491.264,A -85,B 0,C 180,E1 -13619.963,E2 -13619.963} C_VEL
LIN {X 0,Y 359.49,Z 481.841,A -85,B 0,C 180,E1 -13621.388,E2 -13621.388} C_VEL
LIN {X 0,Y 359.426,Z 477.418,A -85,B 0,C 180,E1 -13622.004,E2 -13622.004} C_VEL
LIN {X 0,Y 356.877,Z 467.012,A -85,B 0,C 180,E1 -13623.421,E2 -13623.421} C_VEL
LIN {X 0,Y 355.8,Z 460.605,A -85,B 0,C 180,E1 -13624.143,E2 -13624.143} C_VEL
LIN {X 0,Y 355.841,Z 457.149,A -85,B 0,C 180,E1 -13624.453,E2 -13624.453} C_VEL
LIN {X 0,Y 356.898,Z 444.538,A -85,B 0,C 180,E1 -13625.339,E2 -13625.339} C_VEL
LIN {X 0,Y 357.792,Z 431.557,A -85,B 0,C 180,E1 -13625.973,E2 -13625.973} C_VEL
LIN {X 0,Y 358.265,Z 419.28,A -85,B 0,C 180,E1 -13626.364,E2 -13626.364} C_VEL
LIN {X 0,Y 359.966,Z 343.043,A -85,B 0,C 180,E1 -13627.927,E2 -13627.927} C_VEL
LIN {X 0,Y 357.738,Z 333.866,A -85,B 0,C 180,E1 -13628.317,E2 -13628.317} C_VEL
LIN {X 0,Y 350.383,Z 317.226,A -85,B 0,C 180,E1 -13629.333,E2 -13629.333} C_VEL
LIN {X 0,Y 349.692,Z 315.442,A -85,B 0,C 180,E1 -13629.454,E2 -13629.454} C_VEL
LIN {X 0,Y 347.72,Z 307.174,A -85,B 0,C 180,E1 -13631.929,E2 -13631.929} C_VEL
LIN {X 0,Y 347.692,Z 307.176,A -85,B 0,C 180,E1 -13635.026,E2 -13635.026} C_VEL
LIN {X 0,Y 347.729,Z 307.17,A -85,B 0,C 180,E1 -13638.398,E2 -13638.398} C_VEL
LIN {X 0,Y 347.742,Z 307.17,A -85,B 0,C 180,E1 -13642.677,E2 -13642.677} C_VEL
LIN {X 0,Y 347.735,Z 307.163,A -85,B 0,C 180,E1 -13645.955,E2 -13645.955} C_VEL
LIN {X 0,Y 347.725,Z 307.17,A -85,B 0,C 180,E1 -13649.65,E2 -13649.65} C_VEL
LIN {X 0,Y 347.738,Z 307.171,A -85,B 0,C 180,E1 -13653.6,E2 -13653.6} C_VEL
LIN {X 0,Y 347.756,Z 307.165,A -85,B 0,C 180,E1 -13656.16,E2 -13656.16} C_VEL
LIN {X 0,Y 347.794,Z 307.156,A -85,B 0,C 180,E1 -13659.908,E2 -13659.908} C_VEL
LIN {X 0,Y 347.852,Z 307.149,A -85,B 0,C 180,E1 -13662.359,E2 -13662.359} C_VEL
LIN {X 0,Y 347.884,Z 307.153,A -85,B 0,C 180,E1 -13665.97,E2 -13665.97} C_VEL
LIN {X 0,Y 347.915,Z 307.143,A -85,B 0,C 180,E1 -13669.525,E2 -13669.525} C_VEL
LIN {X 0,Y 348.053,Z 307.118,A -85,B 0,C 180,E1 -13673.042,E2 -13673.042} C_VEL
LIN {X 0,Y 348.192,Z 307.104,A -85,B 0,C 180,E1 -13677.687,E2 -13677.687} C_VEL
LIN {X 0,Y 348.332,Z 307.091,A -85,B 0,C 180,E1 -13680,E2 -13680} C_VEL
LIN {X 0,Y 348.192,Z 307.106,A -85,B 0,C 180,E1 -13682.314,E2 -13682.314} C_VEL
LIN {X 0,Y 348.091,Z 307.12,A -85,B 0,C 180,E1 -13686.958,E2 -13686.958} C_VEL
LIN {X 0,Y 347.915,Z 307.144,A -85,B 0,C 180,E1 -13690.475,E2 -13690.475} C_VEL
LIN {X 0,Y 347.885,Z 307.137,A -85,B 0,C 180,E1 -13694.151,E2 -13694.151} C_VEL
LIN {X 0,Y 347.879,Z 307.144,A -85,B 0,C 180,E1 -13698.291,E2 -13698.291} C_VEL
LIN {X 0,Y 347.776,Z 307.162,A -85,B 0,C 180,E1 -13701.636,E2 -13701.636} C_VEL
LIN {X 0,Y 347.801,Z 307.159,A -85,B 0,C 180,E1 -13705.11,E2 -13705.11} C_VEL
LIN {X 0,Y 347.801,Z 307.152,A -85,B 0,C 180,E1 -13707.695,E2 -13707.695} C_VEL
LIN {X 0,Y 347.76,Z 307.166,A -85,B 0,C 180,E1 -13710.347,E2 -13710.347} C_VEL
LIN {X 0,Y 347.738,Z 307.17,A -85,B 0,C 180,E1 -13714.045,E2 -13714.045} C_VEL
LIN {X 0,Y 347.757,Z 307.17,A -85,B 0,C 180,E1 -13717.322,E2 -13717.322} C_VEL
LIN {X 0,Y 347.747,Z 307.169,A -85,B 0,C 180,E1 -13720.295,E2 -13720.295} C_VEL
LIN {X 0,Y 347.761,Z 307.168,A -85,B 0,C 180,E1 -13723.403,E2 -13723.403} C_VEL
LIN {X 0,Y 347.776,Z 307.154,A -85,B 0,C 180,E1 -13726.678,E2 -13726.678} C_VEL
LIN {X 0,Y 347.779,Z 307.154,A -85,B 0,C 180,E1 -13730.167,E2 -13730.167} C_VEL
LIN {X 0,Y 347.783,Z 307.16,A -85,B 0,C 180,E1 -13734.127,E2 -13734.127} C_VEL
LIN {X 0,Y 347.767,Z 307.205,A -85,B 0,C 180,E1 -13737.473,E2 -13737.473} C_VEL
LIN {X 0,Y 350.724,Z 319.209,A -85,B 0,C 180,E1 -13740.929,E2 -13740.929} C_VEL
LIN {X 0,Y 352.798,Z 329.456,A -85,B 0,C 180,E1 -13743.694,E2 -13743.694} C_VEL
LIN {X 0,Y 352.813,Z 333.307,A -85,B 0,C 180,E1 -13744.644,E2 -13744.644} C_VEL
LIN {X 0,Y 352.199,Z 338.509,A -85,B 0,C 180,E1 -13745.851,E2 -13745.851} C_VEL
LIN {X 0,Y 357.059,Z 362.064,A -85,B 0,C 180,E1 -13746.793,E2 -13746.793} C_VEL
LIN {X 0,Y 359.347,Z 377.694,A -85,B 0,C 180,E1 -13747.325,E2 -13747.325} C_VEL
LIN {X 0,Y 357.691,Z 447.269,A -85,B 0,C 180,E1 -13748.763,E2 -13748.763} C_VEL
LIN {X 0,Y 356.912,Z 461.111,A -85,B 0,C 180,E1 -13749.281,E2 -13749.281} C_VEL
LIN {X 0,Y 355.804,Z 473.013,A -85,B 0,C 180,E1 -13749.93,E2 -13749.93} C_VEL
LIN {X 0,Y 354.619,Z 484.287,A -85,B 0,C 180,E1 -13750.765,E2 -13750.765} C_VEL
LIN {X 0,Y 353.112,Z 495.933,A -85,B 0,C 180,E1 -13751.883,E2 -13751.883} C_VEL
LIN {X 0,Y 351.741,Z 506.411,A -85,B 0,C 180,E1 -13753.161,E2 -13753.161} C_VEL
LIN {X 0,Y 350.435,Z 515.406,A -85,B 0,C 180,E1 -13754.511,E2 -13754.511} C_VEL
LIN {X 0,Y 349.353,Z 523.668,A -85,B 0,C 180,E1 -13756.032,E2 -13756.032} C_VEL
LIN {X 0,Y 348.076,Z 531.301,A -85,B 0,C 180,E1 -13757.762,E2 -13757.762} C_VEL
LIN {X 0,Y 347.275,Z 537.462,A -85,B 0,C 180,E1 -13759.508,E2 -13759.508} C_VEL
LIN {X 0,Y 346.716,Z 542.375,A -85,B 0,C 180,E1 -13761.257,E2 -13761.257} C_VEL
LIN {X 0,Y 346.343,Z 546.181,A -85,B 0,C 180,E1 -13763.009,E2 -13763.009} C_VEL
LIN {X 0,Y 346.229,Z 548.156,A -85,B 0,C 180,E1 -13764.177,E2 -13764.177} C_VEL
LIN {X 0,Y 346.177,Z 549.721,A -85,B 0,C 180,E1 -13765.344,E2 -13765.344} C_VEL
LIN {X 0,Y 346.147,Z 550.845,A -85,B 0,C 180,E1 -13766.51,E2 -13766.51} C_VEL
LIN {X 0,Y 346.161,Z 551.896,A -85,B 0,C 180,E1 -13768.838,E2 -13768.838} C_VEL
LIN {X 0,Y 346.233,Z 551.844,A -85,B 0,C 180,E1 -13770.002,E2 -13770.002} C_VEL
LIN {X 0,Y 346.195,Z 551.368,A -85,B 0,C 180,E1 -13771.165,E2 -13771.165} C_VEL
LIN {X 0,Y 346.168,Z 549.175,A -85,B 0,C 180,E1 -13773.494,E2 -13773.494} C_VEL
LIN {X 0,Y 346.214,Z 545.884,A -85,B 0,C 180,E1 -13775.53,E2 -13775.53} C_VEL
LIN {X 0,Y 346.437,Z 541.105,A -85,B 0,C 180,E1 -13777.579,E2 -13777.579} C_VEL
LIN {X 0,Y 346.822,Z 534.714,A -85,B 0,C 180,E1 -13779.625,E2 -13779.625} C_VEL
LIN {X 0,Y 347.361,Z 527.738,A -85,B 0,C 180,E1 -13781.379,E2 -13781.379} C_VEL
LIN {X 0,Y 348.281,Z 518.994,A -85,B 0,C 180,E1 -13783.123,E2 -13783.123} C_VEL
LIN {X 0,Y 349.24,Z 508.901,A -85,B 0,C 180,E1 -13784.737,E2 -13784.737} C_VEL
LIN {X 0,Y 350.166,Z 498.901,A -85,B 0,C 180,E1 -13786.021,E2 -13786.021} C_VEL
LIN {X 0,Y 351.167,Z 487.635,A -85,B 0,C 180,E1 -13787.171,E2 -13787.171} C_VEL
LIN {X 0,Y 352.195,Z 474.991,A -85,B 0,C 180,E1 -13788.169,E2 -13788.169} C_VEL
LIN {X 0,Y 353.038,Z 462.756,A -85,B 0,C 180,E1 -13788.876,E2 -13788.876} C_VEL
LIN {X 0,Y 353.708,Z 449.204,A -85,B 0,C 180,E1 -13789.403,E2 -13789.403} C_VEL
LIN {X 0,Y 354.32,Z 419.178,A -85,B 0,C 180,E1 -13790.048,E2 -13790.048} C_VEL
LIN {X 0,Y 354.852,Z 374.209,A -85,B 0,C 180,E1 -13790.965,E2 -13790.965} C_VEL
LIN {X 0,Y 350,Z 339.126,A -85,B 0,C 180,E1 -13791.977,E2 -13791.977} C_VEL
LIN {X 0,Y 351.248,Z 324.784,A -85,B 0,C 180,E1 -13795.269,E2 -13795.269} C_VEL
LIN {X 0,Y 349.022,Z 312.811,A -85,B 0,C 180,E1 -13798.256,E2 -13798.256} C_VEL
LIN {X 0,Y 347.829,Z 307.158,A -85,B 0,C 180,E1 -13799.763,E2 -13799.763} C_VEL
LIN {X 0,Y 347.755,Z 307.167,A -85,B 0,C 180,E1 -13804.045,E2 -13804.045} C_VEL
LIN {X 0,Y 347.767,Z 307.162,A -85,B 0,C 180,E1 -13807.322,E2 -13807.322} C_VEL
LIN {X 0,Y 347.739,Z 307.17,A -85,B 0,C 180,E1 -13810.298,E2 -13810.298} C_VEL
LIN {X 0,Y 347.729,Z 307.166,A -85,B 0,C 180,E1 -13813.409,E2 -13813.409} C_VEL
LIN {X 0,Y 347.732,Z 307.173,A -85,B 0,C 180,E1 -13816.687,E2 -13816.687} C_VEL
LIN {X 0,Y 347.754,Z 307.164,A -85,B 0,C 180,E1 -13820.174,E2 -13820.174} C_VEL
LIN {X 0,Y 347.768,Z 307.166,A -85,B 0,C 180,E1 -13822.68,E2 -13822.68} C_VEL
LIN {X 0,Y 347.755,Z 307.163,A -85,B 0,C 180,E1 -13825.957,E2 -13825.957} C_VEL
LIN {X 0,Y 347.771,Z 307.163,A -85,B 0,C 180,E1 -13829.654,E2 -13829.654} C_VEL
LIN {X 0,Y 347.858,Z 307.152,A -85,B 0,C 180,E1 -13832.745,E2 -13832.745} C_VEL
LIN {X 0,Y 347.792,Z 307.159,A -85,B 0,C 180,E1 -13836.162,E2 -13836.162} C_VEL
LIN {X 0,Y 347.806,Z 307.159,A -85,B 0,C 180,E1 -13839.909,E2 -13839.909} C_VEL
LIN {X 0,Y 347.839,Z 307.16,A -85,B 0,C 180,E1 -13843.568,E2 -13843.568} C_VEL
LIN {X 0,Y 347.897,Z 307.147,A -85,B 0,C 180,E1 -13847.161,E2 -13847.161} C_VEL
LIN {X 0,Y 347.947,Z 307.139,A -85,B 0,C 180,E1 -13850.701,E2 -13850.701} C_VEL
LIN {X 0,Y 348.051,Z 307.13,A -85,B 0,C 180,E1 -13854.205,E2 -13854.205} C_VEL
LIN {X 0,Y 348.211,Z 307.109,A -85,B 0,C 180,E1 -13857.686,E2 -13857.686} C_VEL
LIN {X 0,Y 348.329,Z 307.097,A -85,B 0,C 180,E1 -13860,E2 -13860} C_VEL
LIN {X 0,Y 348.211,Z 307.112,A -85,B 0,C 180,E1 -13862.313,E2 -13862.313} C_VEL
LIN {X 0,Y 348.083,Z 307.123,A -85,B 0,C 180,E1 -13866.958,E2 -13866.958} C_VEL
LIN {X 0,Y 347.902,Z 307.151,A -85,B 0,C 180,E1 -13870.475,E2 -13870.475} C_VEL
LIN {X 0,Y 347.905,Z 307.147,A -85,B 0,C 180,E1 -13874.149,E2 -13874.149} C_VEL
LIN {X 0,Y 347.835,Z 307.155,A -85,B 0,C 180,E1 -13878.258,E2 -13878.258} C_VEL
LIN {X 0,Y 347.774,Z 307.161,A -85,B 0,C 180,E1 -13881.626,E2 -13881.626} C_VEL
LIN {X 0,Y 347.817,Z 307.16,A -85,B 0,C 180,E1 -13885.108,E2 -13885.108} C_VEL
LIN {X 0,Y 347.814,Z 307.156,A -85,B 0,C 180,E1 -13887.693,E2 -13887.693} C_VEL
LIN {X 0,Y 347.755,Z 307.164,A -85,B 0,C 180,E1 -13890.347,E2 -13890.347} C_VEL
LIN {X 0,Y 347.753,Z 307.163,A -85,B 0,C 180,E1 -13894.043,E2 -13894.043} C_VEL
LIN {X 0,Y 347.766,Z 307.169,A -85,B 0,C 180,E1 -13897.32,E2 -13897.32} C_VEL
LIN {X 0,Y 347.737,Z 307.165,A -85,B 0,C 180,E1 -13900.296,E2 -13900.296} C_VEL
LIN {X 0,Y 347.728,Z 307.172,A -85,B 0,C 180,E1 -13903.407,E2 -13903.407} C_VEL
LIN {X 0,Y 347.729,Z 307.166,A -85,B 0,C 180,E1 -13906.685,E2 -13906.685} C_VEL
LIN {X 0,Y 347.752,Z 307.166,A -85,B 0,C 180,E1 -13910.172,E2 -13910.172} C_VEL
LIN {X 0,Y 347.765,Z 307.162,A -85,B 0,C 180,E1 -13912.678,E2 -13912.678} C_VEL
LIN {X 0,Y 347.752,Z 307.17,A -85,B 0,C 180,E1 -13915.955,E2 -13915.955} C_VEL
LIN {X 0,Y 347.753,Z 307.166,A -85,B 0,C 180,E1 -13919.651,E2 -13919.651} C_VEL
LIN {X 0,Y 347.834,Z 307.154,A -85,B 0,C 180,E1 -13923.606,E2 -13923.606} C_VEL
LIN {X 0,Y 347.793,Z 307.164,A -85,B 0,C 180,E1 -13926.161,E2 -13926.161} C_VEL
LIN {X 0,Y 347.831,Z 307.155,A -85,B 0,C 180,E1 -13929.909,E2 -13929.909} C_VEL
LIN {X 0,Y 347.87,Z 307.154,A -85,B 0,C 180,E1 -13932.358,E2 -13932.358} C_VEL
LIN {X 0,Y 347.899,Z 307.146,A -85,B 0,C 180,E1 -13935.969,E2 -13935.969} C_VEL
LIN {X 0,Y 347.898,Z 307.145,A -85,B 0,C 180,E1 -13939.523,E2 -13939.523} C_VEL
LIN {X 0,Y 347.992,Z 307.226,A -85,B 0,C 180,E1 -13940.951,E2 -13940.951} C_VEL
LIN {X 0,Y 349.512,Z 315.112,A -85,B 0,C 180,E1 -13943.1,E2 -13943.1} C_VEL
LIN {X 0,Y 352.437,Z 325.414,A -85,B 0,C 180,E1 -13943.475,E2 -13943.475} C_VEL
LIN {X 0,Y 355.4,Z 340.984,A -85,B 0,C 180,E1 -13943.96,E2 -13943.96} C_VEL
LIN {X 0,Y 353.957,Z 422.285,A -85,B 0,C 180,E1 -13945.621,E2 -13945.621} C_VEL
LIN {X 0,Y 353.403,Z 435.541,A -85,B 0,C 180,E1 -13946.114,E2 -13946.114} C_VEL
LIN {X 0,Y 352.799,Z 448.733,A -85,B 0,C 180,E1 -13946.858,E2 -13946.858} C_VEL
LIN {X 0,Y 352.079,Z 459.869,A -85,B 0,C 180,E1 -13947.71,E2 -13947.71} C_VEL
LIN {X 0,Y 351.038,Z 471.482,A -85,B 0,C 180,E1 -13948.851,E2 -13948.851} C_VEL
LIN {X 0,Y 350.008,Z 481.928,A -85,B 0,C 180,E1 -13950.142,E2 -13950.142} C_VEL
LIN {X 0,Y 349.178,Z 490.453,A -85,B 0,C 180,E1 -13951.44,E2 -13951.44} C_VEL
LIN {X 0,Y 348.356,Z 498.322,A -85,B 0,C 180,E1 -13952.889,E2 -13952.889} C_VEL
LIN {X 0,Y 347.619,Z 505.991,A -85,B 0,C 180,E1 -13954.637,E2 -13954.637} C_VEL
LIN {X 0,Y 347.156,Z 512.145,A -85,B 0,C 180,E1 -13956.391,E2 -13956.391} C_VEL
LIN {X 0,Y 346.712,Z 517.047,A -85,B 0,C 180,E1 -13958.156,E2 -13958.156} C_VEL
LIN {X 0,Y 346.381,Z 520.82,A -85,B 0,C 180,E1 -13959.929,E2 -13959.929} C_VEL
LIN {X 0,Y 346.172,Z 523.553,A -85,B 0,C 180,E1 -13961.712,E2 -13961.712} C_VEL
LIN {X 0,Y 346.103,Z 524.854,A -85,B 0,C 180,E1 -13962.918,E2 -13962.918} C_VEL
LIN {X 0,Y 346.036,Z 525.708,A -85,B 0,C 180,E1 -13964.104,E2 -13964.104} C_VEL
LIN {X 0,Y 346,Z 526.125,A -85,B 0,C 180,E1 -13965.309,E2 -13965.309} C_VEL
LIN {X 0,Y 346.114,Z 525.89,A -85,B 0,C 180,E1 -13967.378,E2 -13967.378} C_VEL
LIN {X 0,Y 346.261,Z 524.895,A -85,B 0,C 180,E1 -13968.948,E2 -13968.948} C_VEL
LIN {X 0,Y 346.725,Z 522.186,A -85,B 0,C 180,E1 -13971.188,E2 -13971.188} C_VEL
LIN {X 0,Y 347.281,Z 518.344,A -85,B 0,C 180,E1 -13973.24,E2 -13973.24} C_VEL
LIN {X 0,Y 348.027,Z 513.589,A -85,B 0,C 180,E1 -13975.09,E2 -13975.09} C_VEL
LIN {X 0,Y 348.985,Z 507.427,A -85,B 0,C 180,E1 -13976.941,E2 -13976.941} C_VEL
LIN {X 0,Y 350.247,Z 499.644,A -85,B 0,C 180,E1 -13978.786,E2 -13978.786} C_VEL
LIN {X 0,Y 351.359,Z 492.059,A -85,B 0,C 180,E1 -13980.242,E2 -13980.242} C_VEL
LIN {X 0,Y 352.73,Z 482.663,A -85,B 0,C 180,E1 -13981.711,E2 -13981.711} C_VEL
LIN {X 0,Y 353.999,Z 473.097,A -85,B 0,C 180,E1 -13982.918,E2 -13982.918} C_VEL
LIN {X 0,Y 355.458,Z 461.059,A -85,B 0,C 180,E1 -13984.123,E2 -13984.123} C_VEL
LIN {X 0,Y 355.841,Z 457.149,A -85,B 0,C 180,E1 -13984.453,E2 -13984.453} C_VEL
LIN {X 0,Y 355.69,Z 451.913,A -85,B 0,C 180,E1 -13984.901,E2 -13984.901} C_VEL
LIN {X 0,Y 353.692,Z 443.357,A -85,B 0,C 180,E1 -13985.657,E2 -13985.657} C_VEL
LIN {X 0,Y 351.719,Z 434.542,A -85,B 0,C 180,E1 -13986.307,E2 -13986.307} C_VEL
LIN {X 0,Y 351.503,Z 428.917,A -85,B 0,C 180,E1 -13986.578,E2 -13986.578} C_VEL
LIN {X 0,Y 351.979,Z 416.62,A -85,B 0,C 180,E1 -13986.925,E2 -13986.925} C_VEL
LIN {X 0,Y 353.579,Z 343.842,A -85,B 0,C 180,E1 -13988.442,E2 -13988.442} C_VEL
LIN {X 0,Y 351.788,Z 336.603,A -85,B 0,C 180,E1 -13988.761,E2 -13988.761} C_VEL
LIN {X 0,Y 344.121,Z 319.19,A -85,B 0,C 180,E1 -13989.861,E2 -13989.861} C_VEL
LIN {X 0,Y 342.576,Z 315.725,A -85,B 0,C 180,E1 -13990.113,E2 -13990.113} C_VEL
LIN {X 0,Y 340.713,Z 308.046,A -85,B 0,C 180,E1 -13992.528,E2 -13992.528} C_VEL
LIN {X 0,Y 340.64,Z 308.044,A -85,B 0,C 180,E1 -13996.226,E2 -13996.226} C_VEL
LIN {X 0,Y 340.659,Z 308.051,A -85,B 0,C 180,E1 -13998.687,E2 -13998.687} C_VEL
LIN {X 0,Y 340.706,Z 308.05,A -85,B 0,C 180,E1 -14001.769,E2 -14001.769} C_VEL
LIN {X 0,Y 340.709,Z 308.033,A -85,B 0,C 180,E1 -14005.595,E2 -14005.595} C_VEL
LIN {X 0,Y 340.68,Z 308.043,A -85,B 0,C 180,E1 -14008.954,E2 -14008.954} C_VEL
LIN {X 0,Y 340.708,Z 308.043,A -85,B 0,C 180,E1 -14013.012,E2 -14013.012} C_VEL
LIN {X 0,Y 340.728,Z 308.036,A -85,B 0,C 180,E1 -14015.636,E2 -14015.636} C_VEL
LIN {X 0,Y 340.721,Z 308.034,A -85,B 0,C 180,E1 -14019.473,E2 -14019.473} C_VEL
LIN {X 0,Y 340.844,Z 308.026,A -85,B 0,C 180,E1 -14021.984,E2 -14021.984} C_VEL
LIN {X 0,Y 340.856,Z 308.026,A -85,B 0,C 180,E1 -14025.705,E2 -14025.705} C_VEL
LIN {X 0,Y 340.857,Z 308.021,A -85,B 0,C 180,E1 -14029.306,E2 -14029.306} C_VEL
LIN {X 0,Y 341.001,Z 307.996,A -85,B 0,C 180,E1 -14032.897,E2 -14032.897} C_VEL
LIN {X 0,Y 341.154,Z 307.98,A -85,B 0,C 180,E1 -14037.639,E2 -14037.639} C_VEL
LIN {X 0,Y 341.282,Z 307.969,A -85,B 0,C 180,E1 -14040,E2 -14040} C_VEL
LIN {X 0,Y 341.153,Z 307.982,A -85,B 0,C 180,E1 -14042.362,E2 -14042.362} C_VEL
LIN {X 0,Y 341.061,Z 307.994,A -85,B 0,C 180,E1 -14047.102,E2 -14047.102} C_VEL
LIN {X 0,Y 340.858,Z 308.025,A -85,B 0,C 180,E1 -14050.694,E2 -14050.694} C_VEL
LIN {X 0,Y 340.85,Z 308.014,A -85,B 0,C 180,E1 -14054.326,E2 -14054.326} C_VEL
LIN {X 0,Y 340.825,Z 308.021,A -85,B 0,C 180,E1 -14058.468,E2 -14058.468} C_VEL
LIN {X 0,Y 340.742,Z 308.038,A -85,B 0,C 180,E1 -14061.858,E2 -14061.858} C_VEL
LIN {X 0,Y 340.761,Z 308.038,A -85,B 0,C 180,E1 -14065.666,E2 -14065.666} C_VEL
LIN {X 0,Y 340.731,Z 308.032,A -85,B 0,C 180,E1 -14068.321,E2 -14068.321} C_VEL
LIN {X 0,Y 340.706,Z 308.045,A -85,B 0,C 180,E1 -14071.044,E2 -14071.044} C_VEL
LIN {X 0,Y 340.709,Z 308.043,A -85,B 0,C 180,E1 -14075.28,E2 -14075.28} C_VEL
LIN {X 0,Y 340.71,Z 308.045,A -85,B 0,C 180,E1 -14078.39,E2 -14078.39} C_VEL
LIN {X 0,Y 340.725,Z 308.04,A -85,B 0,C 180,E1 -14082.054,E2 -14082.054} C_VEL
LIN {X 0,Y 340.714,Z 308.031,A -85,B 0,C 180,E1 -14085.47,E2 -14085.47} C_VEL
LIN {X 0,Y 340.729,Z 308.042,A -85,B 0,C 180,E1 -14088.7,E2 -14088.7} C_VEL
LIN {X 0,Y 340.733,Z 308.045,A -85,B 0,C 180,E1 -14091.775,E2 -14091.775} C_VEL
LIN {X 0,Y 340.718,Z 308.044,A -85,B 0,C 180,E1 -14095.597,E2 -14095.597} C_VEL
LIN {X 0,Y 340.729,Z 308.118,A -85,B 0,C 180,E1 -14096.918,E2 -14096.918} C_VEL
LIN {X 0,Y 343.29,Z 318.417,A -85,B 0,C 180,E1 -14099.984,E2 -14099.984} C_VEL
LIN {X 0,Y 345.698,Z 329.582,A -85,B 0,C 180,E1 -14103.109,E2 -14103.109} C_VEL
LIN {X 0,Y 346.138,Z 333.427,A -85,B 0,C 180,E1 -14104.119,E2 -14104.119} C_VEL
LIN {X 0,Y 345.58,Z 338.126,A -85,B 0,C 180,E1 -14105.249,E2 -14105.249} C_VEL
LIN {X 0,Y 350.903,Z 364.042,A -85,B 0,C 180,E1 -14106.324,E2 -14106.324} C_VEL
LIN {X 0,Y 352.983,Z 378.515,A -85,B 0,C 180,E1 -14106.828,E2 -14106.828} C_VEL
LIN {X 0,Y 351.263,Z 447.323,A -85,B 0,C 180,E1 -14108.278,E2 -14108.278} C_VEL
LIN {X 0,Y 350.452,Z 461.052,A -85,B 0,C 180,E1 -14108.804,E2 -14108.804} C_VEL
LIN {X 0,Y 349.194,Z 473.963,A -85,B 0,C 180,E1 -14109.533,E2 -14109.533} C_VEL
LIN {X 0,Y 347.792,Z 486.474,A -85,B 0,C 180,E1 -14110.525,E2 -14110.525} C_VEL
LIN {X 0,Y 346.282,Z 497.653,A -85,B 0,C 180,E1 -14111.666,E2 -14111.666} C_VEL
LIN {X 0,Y 344.773,Z 507.758,A -85,B 0,C 180,E1 -14112.963,E2 -14112.963} C_VEL
LIN {X 0,Y 343.505,Z 516.178,A -85,B 0,C 180,E1 -14114.294,E2 -14114.294} C_VEL
LIN {X 0,Y 342.218,Z 525.119,A -85,B 0,C 180,E1 -14116.038,E2 -14116.038} C_VEL
LIN {X 0,Y 340.972,Z 532.446,A -85,B 0,C 180,E1 -14117.805,E2 -14117.805} C_VEL
LIN {X 0,Y 340.039,Z 539.198,A -85,B 0,C 180,E1 -14119.884,E2 -14119.884} C_VEL
LIN {X 0,Y 339.527,Z 543.68,A -85,B 0,C 180,E1 -14121.671,E2 -14121.671} C_VEL
LIN {X 0,Y 339.274,Z 546.054,A -85,B 0,C 180,E1 -14122.862,E2 -14122.862} C_VEL
LIN {X 0,Y 339.135,Z 548.094,A -85,B 0,C 180,E1 -14124.112,E2 -14124.112} C_VEL
LIN {X 0,Y 339.079,Z 549.542,A -85,B 0,C 180,E1 -14125.246,E2 -14125.246} C_VEL
LIN {X 0,Y 339.071,Z 550.632,A -85,B 0,C 180,E1 -14126.437,E2 -14126.437} C_VEL
LIN {X 0,Y 339.062,Z 551.64,A -85,B 0,C 180,E1 -14128.814,E2 -14128.814} C_VEL
LIN {X 0,Y 339.138,Z 551.565,A -85,B 0,C 180,E1 -14130.002,E2 -14130.002} C_VEL
LIN {X 0,Y 339.097,Z 551.05,A -85,B 0,C 180,E1 -14131.189,E2 -14131.189} C_VEL
LIN {X 0,Y 339.093,Z 548.815,A -85,B 0,C 180,E1 -14133.567,E2 -14133.567} C_VEL
LIN {X 0,Y 339.115,Z 545.81,A -85,B 0,C 180,E1 -14135.462,E2 -14135.462} C_VEL
LIN {X 0,Y 339.27,Z 542.155,A -85,B 0,C 180,E1 -14137.141,E2 -14137.141} C_VEL
LIN {X 0,Y 339.575,Z 537.154,A -85,B 0,C 180,E1 -14138.931,E2 -14138.931} C_VEL
LIN {X 0,Y 340.026,Z 530.849,A -85,B 0,C 180,E1 -14140.722,E2 -14140.722} C_VEL
LIN {X 0,Y 340.794,Z 522.951,A -85,B 0,C 180,E1 -14142.507,E2 -14142.507} C_VEL
LIN {X 0,Y 341.647,Z 514.878,A -85,B 0,C 180,E1 -14143.989,E2 -14143.989} C_VEL
LIN {X 0,Y 342.58,Z 505.003,A -85,B 0,C 180,E1 -14145.469,E2 -14145.469} C_VEL
LIN {X 0,Y 343.588,Z 493.986,A -85,B 0,C 180,E1 -14146.795,E2 -14146.795} C_VEL
LIN {X 0,Y 344.666,Z 483.2,A -85,B 0,C 180,E1 -14147.812,E2 -14147.812} C_VEL
LIN {X 0,Y 345.646,Z 470.174,A -85,B 0,C 180,E1 -14148.756,E2 -14148.756} C_VEL
LIN {X 0,Y 346.478,Z 457.747,A -85,B 0,C 180,E1 -14149.401,E2 -14149.401} C_VEL
LIN {X 0,Y 346.976,Z 444.844,A -85,B 0,C 180,E1 -14149.834,E2 -14149.834} C_VEL
LIN {X 0,Y 348.133,Z 375.463,A -85,B 0,C 180,E1 -14151.275,E2 -14151.275} C_VEL
LIN {X 0,Y 343.11,Z 338.914,A -85,B 0,C 180,E1 -14152.34,E2 -14152.34} C_VEL
LIN {X 0,Y 344.277,Z 325.904,A -85,B 0,C 180,E1 -14155.386,E2 -14155.386} C_VEL
LIN {X 0,Y 341.973,Z 313.527,A -85,B 0,C 180,E1 -14158.545,E2 -14158.545} C_VEL
LIN {X 0,Y 340.765,Z 308.04,A -85,B 0,C 180,E1 -14160.029,E2 -14160.029} C_VEL
LIN {X 0,Y 340.729,Z 308.044,A -85,B 0,C 180,E1 -14164.405,E2 -14164.405} C_VEL
LIN {X 0,Y 340.716,Z 308.047,A -85,B 0,C 180,E1 -14168.387,E2 -14168.387} C_VEL
LIN {X 0,Y 340.705,Z 308.043,A -85,B 0,C 180,E1 -14172.046,E2 -14172.046} C_VEL
LIN {X 0,Y 340.659,Z 308.049,A -85,B 0,C 180,E1 -14176.228,E2 -14176.228} C_VEL
LIN {X 0,Y 340.695,Z 308.043,A -85,B 0,C 180,E1 -14179.754,E2 -14179.754} C_VEL
LIN {X 0,Y 340.711,Z 308.043,A -85,B 0,C 180,E1 -14183.259,E2 -14183.259} C_VEL
LIN {X 0,Y 340.699,Z 308.042,A -85,B 0,C 180,E1 -14186.154,E2 -14186.154} C_VEL
LIN {X 0,Y 340.782,Z 308.032,A -85,B 0,C 180,E1 -14190.333,E2 -14190.333} C_VEL
LIN {X 0,Y 340.811,Z 308.033,A -85,B 0,C 180,E1 -14193.02,E2 -14193.02} C_VEL
LIN {X 0,Y 340.761,Z 308.037,A -85,B 0,C 180,E1 -14195.638,E2 -14195.638} C_VEL
LIN {X 0,Y 340.737,Z 308.043,A -85,B 0,C 180,E1 -14199.473,E2 -14199.473} C_VEL
LIN {X 0,Y 340.799,Z 308.031,A -85,B 0,C 180,E1 -14201.981,E2 -14201.981} C_VEL
LIN {X 0,Y 340.877,Z 308.026,A -85,B 0,C 180,E1 -14205.705,E2 -14205.705} C_VEL
LIN {X 0,Y 340.877,Z 308.022,A -85,B 0,C 180,E1 -14209.306,E2 -14209.306} C_VEL
LIN {X 0,Y 341.01,Z 308.003,A -85,B 0,C 180,E1 -14212.897,E2 -14212.897} C_VEL
LIN {X 0,Y 341.173,Z 307.985,A -85,B 0,C 180,E1 -14217.639,E2 -14217.639} C_VEL
LIN {X 0,Y 341.28,Z 307.975,A -85,B 0,C 180,E1 -14220,E2 -14220} C_VEL
LIN {X 0,Y 341.173,Z 307.987,A -85,B 0,C 180,E1 -14222.361,E2 -14222.361} C_VEL
LIN {X 0,Y 341.051,Z 307.998,A -85,B 0,C 180,E1 -14227.102,E2 -14227.102} C_VEL
LIN {X 0,Y 340.854,Z 308.027,A -85,B 0,C 180,E1 -14230.694,E2 -14230.694} C_VEL
LIN {X 0,Y 340.87,Z 308.025,A -85,B 0,C 180,E1 -14234.324,E2 -14234.324} C_VEL
LIN {X 0,Y 340.791,Z 308.034,A -85,B 0,C 180,E1 -14238.44,E2 -14238.44} C_VEL
LIN {X 0,Y 340.724,Z 308.039,A -85,B 0,C 180,E1 -14241.841,E2 -14241.841} C_VEL
LIN {X 0,Y 340.778,Z 308.033,A -85,B 0,C 180,E1 -14245.664,E2 -14245.664} C_VEL
LIN {X 0,Y 340.734,Z 308.038,A -85,B 0,C 180,E1 -14248.32,E2 -14248.32} C_VEL
LIN {X 0,Y 340.703,Z 308.047,A -85,B 0,C 180,E1 -14251.044,E2 -14251.044} C_VEL
LIN {X 0,Y 340.723,Z 308.046,A -85,B 0,C 180,E1 -14255.278,E2 -14255.278} C_VEL
LIN {X 0,Y 340.714,Z 308.04,A -85,B 0,C 180,E1 -14258.385,E2 -14258.385} C_VEL
LIN {X 0,Y 340.704,Z 308.043,A -85,B 0,C 180,E1 -14262.044,E2 -14262.044} C_VEL
LIN {X 0,Y 340.656,Z 308.048,A -85,B 0,C 180,E1 -14266.226,E2 -14266.226} C_VEL
LIN {X 0,Y 340.693,Z 308.049,A -85,B 0,C 180,E1 -14269.752,E2 -14269.752} C_VEL
LIN {X 0,Y 340.709,Z 308.042,A -85,B 0,C 180,E1 -14273.257,E2 -14273.257} C_VEL
LIN {X 0,Y 340.696,Z 308.047,A -85,B 0,C 180,E1 -14276.152,E2 -14276.152} C_VEL
LIN {X 0,Y 340.745,Z 308.04,A -85,B 0,C 180,E1 -14280.328,E2 -14280.328} C_VEL
LIN {X 0,Y 340.807,Z 308.029,A -85,B 0,C 180,E1 -14283.019,E2 -14283.019} C_VEL
LIN {X 0,Y 340.734,Z 308.039,A -85,B 0,C 180,E1 -14286.926,E2 -14286.926} C_VEL
LIN {X 0,Y 340.803,Z 308.033,A -85,B 0,C 180,E1 -14290.733,E2 -14290.733} C_VEL
LIN {X 0,Y 340.789,Z 308.031,A -85,B 0,C 180,E1 -14293.217,E2 -14293.217} C_VEL
LIN {X 0,Y 340.846,Z 308.027,A -85,B 0,C 180,E1 -14296.889,E2 -14296.889} C_VEL
LIN {X 0,Y 340.91,Z 308.16,A -85,B 0,C 180,E1 -14300.701,E2 -14300.701} C_VEL
LIN {X 0,Y 342.354,Z 315.312,A -85,B 0,C 180,E1 -14302.701,E2 -14302.701} C_VEL
LIN {X 0,Y 345.739,Z 326.671,A -85,B 0,C 180,E1 -14303.143,E2 -14303.143} C_VEL
LIN {X 0,Y 348.659,Z 342.132,A -85,B 0,C 180,E1 -14303.633,E2 -14303.633} C_VEL
LIN {X 0,Y 347.119,Z 423.116,A -85,B 0,C 180,E1 -14305.324,E2 -14305.324} C_VEL
LIN {X 0,Y 346.54,Z 436.777,A -85,B 0,C 180,E1 -14305.855,E2 -14305.855} C_VEL
LIN {X 0,Y 345.925,Z 449.16,A -85,B 0,C 180,E1 -14306.577,E2 -14306.577} C_VEL
LIN {X 0,Y 345.122,Z 461.039,A -85,B 0,C 180,E1 -14307.518,E2 -14307.518} C_VEL
LIN {X 0,Y 344.063,Z 472.414,A -85,B 0,C 180,E1 -14308.673,E2 -14308.673} C_VEL
LIN {X 0,Y 343.005,Z 482.8,A -85,B 0,C 180,E1 -14309.998,E2 -14309.998} C_VEL
LIN {X 0,Y 342.055,Z 492.041,A -85,B 0,C 180,E1 -14311.47,E2 -14311.47} C_VEL
LIN {X 0,Y 341.088,Z 501.03,A -85,B 0,C 180,E1 -14313.246,E2 -14313.246} C_VEL
LIN {X 0,Y 340.369,Z 508.265,A -85,B 0,C 180,E1 -14315.033,E2 -14315.033} C_VEL
LIN {X 0,Y 339.913,Z 514.631,A -85,B 0,C 180,E1 -14317.051,E2 -14317.051} C_VEL
LIN {X 0,Y 339.477,Z 519.197,A -85,B 0,C 180,E1 -14318.93,E2 -14318.93} C_VEL
LIN {X 0,Y 339.15,Z 522.483,A -85,B 0,C 180,E1 -14320.747,E2 -14320.747} C_VEL
LIN {X 0,Y 338.997,Z 525.161,A -85,B 0,C 180,E1 -14322.996,E2 -14322.996} C_VEL
LIN {X 0,Y 338.929,Z 526.075,A -85,B 0,C 180,E1 -14324.406,E2 -14324.406} C_VEL
LIN {X 0,Y 338.904,Z 526.428,A -85,B 0,C 180,E1 -14325.638,E2 -14325.638} C_VEL
LIN {X 0,Y 339.035,Z 526.148,A -85,B 0,C 180,E1 -14327.532,E2 -14327.532} C_VEL
LIN {X 0,Y 339.242,Z 524.935,A -85,B 0,C 180,E1 -14329.356,E2 -14329.356} C_VEL
LIN {X 0,Y 339.682,Z 522.445,A -85,B 0,C 180,E1 -14331.402,E2 -14331.402} C_VEL
LIN {X 0,Y 340.182,Z 519.391,A -85,B 0,C 180,E1 -14333.11,E2 -14333.11} C_VEL
LIN {X 0,Y 340.971,Z 514.517,A -85,B 0,C 180,E1 -14335.138,E2 -14335.138} C_VEL
LIN {X 0,Y 341.878,Z 509.064,A -85,B 0,C 180,E1 -14336.886,E2 -14336.886} C_VEL
LIN {X 0,Y 343.153,Z 501.634,A -85,B 0,C 180,E1 -14338.768,E2 -14338.768} C_VEL
LIN {X 0,Y 344.382,Z 493.944,A -85,B 0,C 180,E1 -14340.335,E2 -14340.335} C_VEL
LIN {X 0,Y 345.856,Z 484.52,A -85,B 0,C 180,E1 -14341.891,E2 -14341.891} C_VEL
LIN {X 0,Y 347.33,Z 474.078,A -85,B 0,C 180,E1 -14343.274,E2 -14343.274} C_VEL
LIN {X 0,Y 348.842,Z 462.08,A -85,B 0,C 180,E1 -14344.513,E2 -14344.513} C_VEL
LIN {X 0,Y 349.961,Z 450.588,A -85,B 0,C 180,E1 -14345.439,E2 -14345.439} C_VEL
LIN {X 0,Y 350.921,Z 439.243,A -85,B 0,C 180,E1 -14346.123,E2 -14346.123} C_VEL
LIN {X 0,Y 351.503,Z 428.917,A -85,B 0,C 180,E1 -14346.578,E2 -14346.578} C_VEL
LIN {X 0,Y 351.293,Z 423.196,A -85,B 0,C 180,E1 -14346.814,E2 -14346.814} C_VEL
LIN {X 0,Y 348.989,Z 413.926,A -85,B 0,C 180,E1 -14347.255,E2 -14347.255} C_VEL
LIN {X 0,Y 346.525,Z 404.595,A -85,B 0,C 180,E1 -14347.655,E2 -14347.655} C_VEL
LIN {X 0,Y 346.066,Z 398.777,A -85,B 0,C 180,E1 -14347.819,E2 -14347.819} C_VEL
LIN {X 0,Y 347.329,Z 345.193,A -85,B 0,C 180,E1 -14348.955,E2 -14348.955} C_VEL
LIN {X 0,Y 345.883,Z 339.465,A -85,B 0,C 180,E1 -14349.219,E2 -14349.219} C_VEL
LIN {X 0,Y 338.58,Z 322.816,A -85,B 0,C 180,E1 -14350.303,E2 -14350.303} C_VEL
LIN {X 0,Y 335.412,Z 316.058,A -85,B 0,C 180,E1 -14350.8,E2 -14350.8} C_VEL
LIN {X 0,Y 333.616,Z 308.93,A -85,B 0,C 180,E1 -14353.122,E2 -14353.122} C_VEL
LIN {X 0,Y 333.617,Z 308.927,A -85,B 0,C 180,E1 -14357.499,E2 -14357.499} C_VEL
LIN {X 0,Y 333.604,Z 308.93,A -85,B 0,C 180,E1 -14361.209,E2 -14361.209} C_VEL
LIN {X 0,Y 333.661,Z 308.906,A -85,B 0,C 180,E1 -14363.859,E2 -14363.859} C_VEL
LIN {X 0,Y 333.631,Z 308.93,A -85,B 0,C 180,E1 -14367.412,E2 -14367.412} C_VEL
LIN {X 0,Y 333.64,Z 308.924,A -85,B 0,C 180,E1 -14371.021,E2 -14371.021} C_VEL
LIN {X 0,Y 333.683,Z 308.913,A -85,B 0,C 180,E1 -14375.087,E2 -14375.087} C_VEL
LIN {X 0,Y 333.66,Z 308.913,A -85,B 0,C 180,E1 -14379.018,E2 -14379.018} C_VEL
LIN {X 0,Y 333.78,Z 308.908,A -85,B 0,C 180,E1 -14381.589,E2 -14381.589} C_VEL
LIN {X 0,Y 333.795,Z 308.905,A -85,B 0,C 180,E1 -14385.576,E2 -14385.576} C_VEL
LIN {X 0,Y 333.82,Z 308.898,A -85,B 0,C 180,E1 -14389.078,E2 -14389.078} C_VEL
LIN {X 0,Y 333.954,Z 308.874,A -85,B 0,C 180,E1 -14392.746,E2 -14392.746} C_VEL
LIN {X 0,Y 333.789,Z 308.905,A -85,B 0,C 180,E1 -14395.169,E2 -14395.169} C_VEL
LIN {X 0,Y 334.091,Z 308.86,A -85,B 0,C 180,E1 -14397.589,E2 -14397.589} C_VEL
LIN {X 0,Y 334.233,Z 308.847,A -85,B 0,C 180,E1 -14400,E2 -14400} C_VEL
LIN {X 0,Y 334.091,Z 308.86,A -85,B 0,C 180,E1 -14402.412,E2 -14402.412} C_VEL
LIN {X 0,Y 334.01,Z 308.872,A -85,B 0,C 180,E1 -14407.253,E2 -14407.253} C_VEL
LIN {X 0,Y 333.821,Z 308.904,A -85,B 0,C 180,E1 -14410.923,E2 -14410.923} C_VEL
LIN {X 0,Y 333.795,Z 308.895,A -85,B 0,C 180,E1 -14414.635,E2 -14414.635} C_VEL
LIN {X 0,Y 333.784,Z 308.897,A -85,B 0,C 180,E1 -14418.656,E2 -14418.656} C_VEL
LIN {X 0,Y 333.68,Z 308.918,A -85,B 0,C 180,E1 -14422.279,E2 -14422.279} C_VEL
LIN {X 0,Y 333.725,Z 308.913,A -85,B 0,C 180,E1 -14426.248,E2 -14426.248} C_VEL
LIN {X 0,Y 333.701,Z 308.911,A -85,B 0,C 180,E1 -14428.973,E2 -14428.973} C_VEL
LIN {X 0,Y 333.641,Z 308.918,A -85,B 0,C 180,E1 -14432.591,E2 -14432.591} C_VEL
LIN {X 0,Y 333.668,Z 308.918,A -85,B 0,C 180,E1 -14436.14,E2 -14436.14} C_VEL
LIN {X 0,Y 333.664,Z 308.921,A -85,B 0,C 180,E1 -14439.19,E2 -14439.19} C_VEL
LIN {X 0,Y 333.668,Z 308.919,A -85,B 0,C 180,E1 -14442.51,E2 -14442.51} C_VEL
LIN {X 0,Y 333.66,Z 308.908,A -85,B 0,C 180,E1 -14445.969,E2 -14445.969} C_VEL
LIN {X 0,Y 333.696,Z 308.912,A -85,B 0,C 180,E1 -14449.306,E2 -14449.306} C_VEL
LIN {X 0,Y 333.66,Z 308.918,A -85,B 0,C 180,E1 -14453.17,E2 -14453.17} C_VEL
LIN {X 0,Y 333.684,Z 309.08,A -85,B 0,C 180,E1 -14456.348,E2 -14456.348} C_VEL
LIN {X 0,Y 336.135,Z 318.851,A -85,B 0,C 180,E1 -14459.348,E2 -14459.348} C_VEL
LIN {X 0,Y 338.309,Z 328.451,A -85,B 0,C 180,E1 -14462.136,E2 -14462.136} C_VEL
LIN {X 0,Y 339.313,Z 334.996,A -85,B 0,C 180,E1 -14463.93,E2 -14463.93} C_VEL
LIN {X 0,Y 338.939,Z 337.932,A -85,B 0,C 180,E1 -14464.632,E2 -14464.632} C_VEL
LIN {X 0,Y 344.421,Z 364.163,A -85,B 0,C 180,E1 -14465.763,E2 -14465.763} C_VEL
LIN {X 0,Y 346.582,Z 377.837,A -85,B 0,C 180,E1 -14466.272,E2 -14466.272} C_VEL
LIN {X 0,Y 344.873,Z 447.372,A -85,B 0,C 180,E1 -14467.775,E2 -14467.775} C_VEL
LIN {X 0,Y 344.018,Z 460.998,A -85,B 0,C 180,E1 -14468.309,E2 -14468.309} C_VEL
LIN {X 0,Y 342.831,Z 472.78,A -85,B 0,C 180,E1 -14468.979,E2 -14468.979} C_VEL
LIN {X 0,Y 341.538,Z 483.961,A -85,B 0,C 180,E1 -14469.84,E2 -14469.84} C_VEL
LIN {X 0,Y 339.867,Z 495.556,A -85,B 0,C 180,E1 -14470.995,E2 -14470.995} C_VEL
LIN {X 0,Y 338.35,Z 505.996,A -85,B 0,C 180,E1 -14472.317,E2 -14472.317} C_VEL
LIN {X 0,Y 336.835,Z 514.872,A -85,B 0,C 180,E1 -14473.697,E2 -14473.697} C_VEL
LIN {X 0,Y 335.838,Z 522.467,A -85,B 0,C 180,E1 -14475.148,E2 -14475.148} C_VEL
LIN {X 0,Y 334.414,Z 530.25,A -85,B 0,C 180,E1 -14476.945,E2 -14476.945} C_VEL
LIN {X 0,Y 333.517,Z 535.565,A -85,B 0,C 180,E1 -14478.454,E2 -14478.454} C_VEL
LIN {X 0,Y 332.803,Z 540.768,A -85,B 0,C 180,E1 -14480.276,E2 -14480.276} C_VEL
LIN {X 0,Y 332.357,Z 544.83,A -85,B 0,C 180,E1 -14482.102,E2 -14482.102} C_VEL
LIN {X 0,Y 332.031,Z 548.204,A -85,B 0,C 180,E1 -14484.178,E2 -14484.178} C_VEL
LIN {X 0,Y 331.997,Z 550.419,A -85,B 0,C 180,E1 -14486.361,E2 -14486.361} C_VEL
LIN {X 0,Y 331.965,Z 551.385,A -85,B 0,C 180,E1 -14488.789,E2 -14488.789} C_VEL
LIN {X 0,Y 332.043,Z 551.277,A -85,B 0,C 180,E1 -14490.002,E2 -14490.002} C_VEL
LIN {X 0,Y 332,Z 550.731,A -85,B 0,C 180,E1 -14491.215,E2 -14491.215} C_VEL
LIN {X 0,Y 332.018,Z 548.454,A -85,B 0,C 180,E1 -14493.643,E2 -14493.643} C_VEL
LIN {X 0,Y 332.018,Z 546.676,A -85,B 0,C 180,E1 -14494.859,E2 -14494.859} C_VEL
LIN {X 0,Y 332.159,Z 543.141,A -85,B 0,C 180,E1 -14496.684,E2 -14496.684} C_VEL
LIN {X 0,Y 332.385,Z 538.477,A -85,B 0,C 180,E1 -14498.513,E2 -14498.513} C_VEL
LIN {X 0,Y 332.933,Z 531.416,A -85,B 0,C 180,E1 -14500.646,E2 -14500.646} C_VEL
LIN {X 0,Y 333.657,Z 523.761,A -85,B 0,C 180,E1 -14502.47,E2 -14502.47} C_VEL
LIN {X 0,Y 334.502,Z 515.924,A -85,B 0,C 180,E1 -14503.984,E2 -14503.984} C_VEL
LIN {X 0,Y 335.493,Z 506.271,A -85,B 0,C 180,E1 -14505.501,E2 -14505.501} C_VEL
LIN {X 0,Y 336.528,Z 495.666,A -85,B 0,C 180,E1 -14506.845,E2 -14506.845} C_VEL
LIN {X 0,Y 337.521,Z 485.395,A -85,B 0,C 180,E1 -14507.888,E2 -14507.888} C_VEL
LIN {X 0,Y 338.533,Z 473.237,A -85,B 0,C 180,E1 -14508.851,E2 -14508.851} C_VEL
LIN {X 0,Y 339.561,Z 459.719,A -85,B 0,C 180,E1 -14509.616,E2 -14509.616} C_VEL
LIN {X 0,Y 340.106,Z 447.177,A -85,B 0,C 180,E1 -14510.094,E2 -14510.094} C_VEL
LIN {X 0,Y 341.368,Z 376.243,A -85,B 0,C 180,E1 -14511.607,E2 -14511.607} C_VEL
LIN {X 0,Y 336.221,Z 338.56,A -85,B 0,C 180,E1 -14512.751,E2 -14512.751} C_VEL
LIN {X 0,Y 337.287,Z 327.928,A -85,B 0,C 180,E1 -14515.289,E2 -14515.289} C_VEL
LIN {X 0,Y 336.215,Z 321.028,A -85,B 0,C 180,E1 -14517.057,E2 -14517.057} C_VEL
LIN {X 0,Y 333.781,Z 309.326,A -85,B 0,C 180,E1 -14520.17,E2 -14520.17} C_VEL
LIN {X 0,Y 333.704,Z 308.92,A -85,B 0,C 180,E1 -14520.363,E2 -14520.363} C_VEL
LIN {X 0,Y 333.692,Z 308.917,A -85,B 0,C 180,E1 -14524.775,E2 -14524.775} C_VEL
LIN {X 0,Y 333.658,Z 308.92,A -85,B 0,C 180,E1 -14527.652,E2 -14527.652} C_VEL
LIN {X 0,Y 333.653,Z 308.924,A -85,B 0,C 180,E1 -14530.768,E2 -14530.768} C_VEL
LIN {X 0,Y 333.6,Z 308.93,A -85,B 0,C 180,E1 -14534.251,E2 -14534.251} C_VEL
LIN {X 0,Y 333.648,Z 308.921,A -85,B 0,C 180,E1 -14537.619,E2 -14537.619} C_VEL
LIN {X 0,Y 333.659,Z 308.922,A -85,B 0,C 180,E1 -14541.203,E2 -14541.203} C_VEL
LIN {X 0,Y 333.682,Z 308.916,A -85,B 0,C 180,E1 -14543.861,E2 -14543.861} C_VEL
LIN {X 0,Y 333.65,Z 308.923,A -85,B 0,C 180,E1 -14547.414,E2 -14547.414} C_VEL
LIN {X 0,Y 333.718,Z 308.917,A -85,B 0,C 180,E1 -14551.028,E2 -14551.028} C_VEL
LIN {X 0,Y 333.742,Z 308.91,A -85,B 0,C 180,E1 -14553.754,E2 -14553.754} C_VEL
LIN {X 0,Y 333.664,Z 308.921,A -85,B 0,C 180,E1 -14557.719,E2 -14557.719} C_VEL
LIN {X 0,Y 333.748,Z 308.912,A -85,B 0,C 180,E1 -14561.587,E2 -14561.587} C_VEL
LIN {X 0,Y 333.815,Z 308.905,A -85,B 0,C 180,E1 -14565.577,E2 -14565.577} C_VEL
LIN {X 0,Y 333.84,Z 308.897,A -85,B 0,C 180,E1 -14569.078,E2 -14569.078} C_VEL
LIN {X 0,Y 333.965,Z 308.879,A -85,B 0,C 180,E1 -14572.746,E2 -14572.746} C_VEL
LIN {X 0,Y 333.805,Z 308.9,A -85,B 0,C 180,E1 -14575.169,E2 -14575.169} C_VEL
LIN {X 0,Y 334.11,Z 308.865,A -85,B 0,C 180,E1 -14577.589,E2 -14577.589} C_VEL
LIN {X 0,Y 334.232,Z 308.853,A -85,B 0,C 180,E1 -14580,E2 -14580} C_VEL
LIN {X 0,Y 334.11,Z 308.866,A -85,B 0,C 180,E1 -14582.411,E2 -14582.411} C_VEL
LIN {X 0,Y 333.987,Z 308.876,A -85,B 0,C 180,E1 -14586.61,E2 -14586.61} C_VEL
LIN {X 0,Y 333.827,Z 308.898,A -85,B 0,C 180,E1 -14589.696,E2 -14589.696} C_VEL
LIN {X 0,Y 333.803,Z 308.901,A -85,B 0,C 180,E1 -14593.391,E2 -14593.391} C_VEL
LIN {X 0,Y 333.725,Z 308.913,A -85,B 0,C 180,E1 -14597.147,E2 -14597.147} C_VEL
LIN {X 0,Y 333.677,Z 308.917,A -85,B 0,C 180,E1 -14599.694,E2 -14599.694} C_VEL
LIN {X 0,Y 333.675,Z 308.917,A -85,B 0,C 180,E1 -14603.59,E2 -14603.59} C_VEL
LIN {X 0,Y 333.74,Z 308.909,A -85,B 0,C 180,E1 -14606.246,E2 -14606.246} C_VEL
LIN {X 0,Y 333.696,Z 308.92,A -85,B 0,C 180,E1 -14608.973,E2 -14608.973} C_VEL
LIN {X 0,Y 333.649,Z 308.921,A -85,B 0,C 180,E1 -14612.586,E2 -14612.586} C_VEL
LIN {X 0,Y 333.681,Z 308.916,A -85,B 0,C 180,E1 -14616.138,E2 -14616.138} C_VEL
LIN {X 0,Y 333.651,Z 308.924,A -85,B 0,C 180,E1 -14619.191,E2 -14619.191} C_VEL
LIN {X 0,Y 333.637,Z 308.922,A -85,B 0,C 180,E1 -14622.499,E2 -14622.499} C_VEL
LIN {X 0,Y 333.601,Z 308.929,A -85,B 0,C 180,E1 -14625.954,E2 -14625.954} C_VEL
LIN {X 0,Y 333.652,Z 308.922,A -85,B 0,C 180,E1 -14629.314,E2 -14629.314} C_VEL
LIN {X 0,Y 333.669,Z 308.919,A -85,B 0,C 180,E1 -14633.167,E2 -14633.167} C_VEL
LIN {X 0,Y 333.678,Z 308.918,A -85,B 0,C 180,E1 -14635.34,E2 -14635.34} C_VEL
LIN {X 0,Y 333.694,Z 308.917,A -85,B 0,C 180,E1 -14639.636,E2 -14639.636} C_VEL
LIN {X 0,Y 333.743,Z 308.913,A -85,B 0,C 180,E1 -14642.399,E2 -14642.399} C_VEL
LIN {X 0,Y 333.73,Z 308.911,A -85,B 0,C 180,E1 -14645.089,E2 -14645.089} C_VEL
LIN {X 0,Y 333.697,Z 308.915,A -85,B 0,C 180,E1 -14649.019,E2 -14649.019} C_VEL
LIN {X 0,Y 333.798,Z 308.902,A -85,B 0,C 180,E1 -14651.588,E2 -14651.588} C_VEL
LIN {X 0,Y 333.81,Z 308.901,A -85,B 0,C 180,E1 -14655.575,E2 -14655.575} C_VEL
LIN {X 0,Y 333.819,Z 308.902,A -85,B 0,C 180,E1 -14659.076,E2 -14659.076} C_VEL
LIN {X 0,Y 333.853,Z 308.984,A -85,B 0,C 180,E1 -14660.416,E2 -14660.416} C_VEL
LIN {X 0,Y 335.204,Z 315.594,A -85,B 0,C 180,E1 -14662.302,E2 -14662.302} C_VEL
LIN {X 0,Y 339.121,Z 328.208,A -85,B 0,C 180,E1 -14662.81,E2 -14662.81} C_VEL
LIN {X 0,Y 341.804,Z 342.381,A -85,B 0,C 180,E1 -14663.271,E2 -14663.271} C_VEL
LIN {X 0,Y 340.294,Z 423.529,A -85,B 0,C 180,E1 -14665.004,E2 -14665.004} C_VEL
LIN {X 0,Y 339.714,Z 437.194,A -85,B 0,C 180,E1 -14665.549,E2 -14665.549} C_VEL
LIN {X 0,Y 339.059,Z 449.545,A -85,B 0,C 180,E1 -14666.284,E2 -14666.284} C_VEL
LIN {X 0,Y 338.169,Z 462.185,A -85,B 0,C 180,E1 -14667.318,E2 -14667.318} C_VEL
LIN {X 0,Y 337.109,Z 473.214,A -85,B 0,C 180,E1 -14668.475,E2 -14668.475} C_VEL
LIN {X 0,Y 336.013,Z 483.629,A -85,B 0,C 180,E1 -14669.848,E2 -14669.848} C_VEL
LIN {X 0,Y 334.932,Z 493.588,A -85,B 0,C 180,E1 -14671.501,E2 -14671.501} C_VEL
LIN {X 0,Y 333.968,Z 502.358,A -85,B 0,C 180,E1 -14673.316,E2 -14673.316} C_VEL
LIN {X 0,Y 333.223,Z 509.347,A -85,B 0,C 180,E1 -14675.141,E2 -14675.141} C_VEL
LIN {X 0,Y 332.816,Z 515.074,A -85,B 0,C 180,E1 -14677.028,E2 -14677.028} C_VEL
LIN {X 0,Y 332.348,Z 519.961,A -85,B 0,C 180,E1 -14679.124,E2 -14679.124} C_VEL
LIN {X 0,Y 332.046,Z 523.108,A -85,B 0,C 180,E1 -14680.98,E2 -14680.98} C_VEL
LIN {X 0,Y 331.907,Z 525.477,A -85,B 0,C 180,E1 -14683.086,E2 -14683.086} C_VEL
LIN {X 0,Y 331.825,Z 526.442,A -85,B 0,C 180,E1 -14684.722,E2 -14684.722} C_VEL
LIN {X 0,Y 331.829,Z 526.731,A -85,B 0,C 180,E1 -14685.98,E2 -14685.98} C_VEL
LIN {X 0,Y 331.975,Z 526.401,A -85,B 0,C 180,E1 -14687.7,E2 -14687.7} C_VEL
LIN {X 0,Y 332.231,Z 524.975,A -85,B 0,C 180,E1 -14689.781,E2 -14689.781} C_VEL
LIN {X 0,Y 332.655,Z 522.699,A -85,B 0,C 180,E1 -14691.63,E2 -14691.63} C_VEL
LIN {X 0,Y 333.257,Z 519.153,A -85,B 0,C 180,E1 -14693.619,E2 -14693.619} C_VEL
LIN {X 0,Y 334.119,Z 514.333,A -85,B 0,C 180,E1 -14695.607,E2 -14695.607} C_VEL
LIN {X 0,Y 335.151,Z 508.464,A -85,B 0,C 180,E1 -14697.471,E2 -14697.471} C_VEL
LIN {X 0,Y 336.554,Z 500.8,A -85,B 0,C 180,E1 -14699.386,E2 -14699.386} C_VEL
LIN {X 0,Y 337.884,Z 492.885,A -85,B 0,C 180,E1 -14700.982,E2 -14700.982} C_VEL
LIN {X 0,Y 339.44,Z 483.15,A -85,B 0,C 180,E1 -14702.567,E2 -14702.567} C_VEL
LIN {X 0,Y 341.028,Z 472.482,A -85,B 0,C 180,E1 -14703.94,E2 -14703.94} C_VEL
LIN {X 0,Y 342.433,Z 461.43,A -85,B 0,C 180,E1 -14705.073,E2 -14705.073} C_VEL
LIN {X 0,Y 343.622,Z 449.662,A -85,B 0,C 180,E1 -14706.014,E2 -14706.014} C_VEL
LIN {X 0,Y 344.66,Z 436.962,A -85,B 0,C 180,E1 -14706.749,E2 -14706.749} C_VEL
LIN {X 0,Y 345.348,Z 424.07,A -85,B 0,C 180,E1 -14707.257,E2 -14707.257} C_VEL
LIN {X 0,Y 346.066,Z 398.777,A -85,B 0,C 180,E1 -14707.819,E2 -14707.819} C_VEL
LIN {X 0,Y 345.642,Z 392.974,A -85,B 0,C 180,E1 -14707.99,E2 -14707.99} C_VEL
LIN {X 0,Y 340.997,Z 374.357,A -85,B 0,C 180,E1 -14708.839,E2 -14708.839} C_VEL
LIN {X 0,Y 340.604,Z 368.554,A -85,B 0,C 180,E1 -14709.013,E2 -14709.013} C_VEL
LIN {X 0,Y 341.104,Z 346.53,A -85,B 0,C 180,E1 -14709.492,E2 -14709.492} C_VEL
LIN {X 0,Y 339.845,Z 341.866,A -85,B 0,C 180,E1 -14709.722,E2 -14709.722} C_VEL
LIN {X 0,Y 332.961,Z 326.226,A -85,B 0,C 180,E1 -14710.779,E2 -14710.779} C_VEL
LIN {X 0,Y 328.208,Z 316.299,A -85,B 0,C 180,E1 -14711.562,E2 -14711.562} C_VEL
LIN {X 0,Y 326.558,Z 309.809,A -85,B 0,C 180,E1 -14713.711,E2 -14713.711} C_VEL
LIN {X 0,Y 326.562,Z 309.801,A -85,B 0,C 180,E1 -14717.027,E2 -14717.027} C_VEL
LIN {X 0,Y 326.559,Z 309.807,A -85,B 0,C 180,E1 -14720.78,E2 -14720.78} C_VEL
LIN {X 0,Y 326.598,Z 309.783,A -85,B 0,C 180,E1 -14724.479,E2 -14724.479} C_VEL
LIN {X 0,Y 326.595,Z 309.806,A -85,B 0,C 180,E1 -14727.454,E2 -14727.454} C_VEL
LIN {X 0,Y 326.603,Z 309.802,A -85,B 0,C 180,E1 -14730.335,E2 -14730.335} C_VEL
LIN {X 0,Y 326.628,Z 309.793,A -85,B 0,C 180,E1 -14734.644,E2 -14734.644} C_VEL
LIN {X 0,Y 326.606,Z 309.793,A -85,B 0,C 180,E1 -14738.543,E2 -14738.543} C_VEL
LIN {X 0,Y 326.731,Z 309.785,A -85,B 0,C 180,E1 -14741.177,E2 -14741.177} C_VEL
LIN {X 0,Y 326.749,Z 309.782,A -85,B 0,C 180,E1 -14745.433,E2 -14745.433} C_VEL
LIN {X 0,Y 326.756,Z 309.776,A -85,B 0,C 180,E1 -14748.839,E2 -14748.839} C_VEL
LIN {X 0,Y 326.908,Z 309.752,A -85,B 0,C 180,E1 -14752.589,E2 -14752.589} C_VEL
LIN {X 0,Y 326.756,Z 309.781,A -85,B 0,C 180,E1 -14755.065,E2 -14755.065} C_VEL
LIN {X 0,Y 327.031,Z 309.739,A -85,B 0,C 180,E1 -14757.537,E2 -14757.537} C_VEL
LIN {X 0,Y 327.184,Z 309.725,A -85,B 0,C 180,E1 -14760,E2 -14760} C_VEL
LIN {X 0,Y 327.031,Z 309.738,A -85,B 0,C 180,E1 -14762.464,E2 -14762.464} C_VEL
LIN {X 0,Y 326.981,Z 309.753,A -85,B 0,C 180,E1 -14766.17,E2 -14766.17} C_VEL
LIN {X 0,Y 326.901,Z 309.752,A -85,B 0,C 180,E1 -14768.656,E2 -14768.656} C_VEL
LIN {X 0,Y 326.722,Z 309.783,A -85,B 0,C 180,E1 -14772.422,E2 -14772.422} C_VEL
LIN {X 0,Y 326.741,Z 309.778,A -85,B 0,C 180,E1 -14774.958,E2 -14774.958} C_VEL
LIN {X 0,Y 326.721,Z 309.777,A -85,B 0,C 180,E1 -14778.84,E2 -14778.84} C_VEL
LIN {X 0,Y 326.609,Z 309.795,A -85,B 0,C 180,E1 -14782.789,E2 -14782.789} C_VEL
LIN {X 0,Y 326.679,Z 309.794,A -85,B 0,C 180,E1 -14785.485,E2 -14785.485} C_VEL
LIN {X 0,Y 326.651,Z 309.797,A -85,B 0,C 180,E1 -14789.66,E2 -14789.66} C_VEL
LIN {X 0,Y 326.613,Z 309.796,A -85,B 0,C 180,E1 -14792.949,E2 -14792.949} C_VEL
LIN {X 0,Y 326.624,Z 309.8,A -85,B 0,C 180,E1 -14797.048,E2 -14797.048} C_VEL
LIN {X 0,Y 326.595,Z 309.805,A -85,B 0,C 180,E1 -14800.209,E2 -14800.209} C_VEL
LIN {X 0,Y 326.602,Z 309.805,A -85,B 0,C 180,E1 -14803.519,E2 -14803.519} C_VEL
LIN {X 0,Y 326.622,Z 309.791,A -85,B 0,C 180,E1 -14807.02,E2 -14807.02} C_VEL
LIN {X 0,Y 326.639,Z 309.789,A -85,B 0,C 180,E1 -14810.768,E2 -14810.768} C_VEL
LIN {X 0,Y 326.607,Z 309.8,A -85,B 0,C 180,E1 -14814.482,E2 -14814.482} C_VEL
LIN {X 0,Y 326.647,Z 309.922,A -85,B 0,C 180,E1 -14815.709,E2 -14815.709} C_VEL
LIN {X 0,Y 329.012,Z 319.344,A -85,B 0,C 180,E1 -14818.698,E2 -14818.698} C_VEL
LIN {X 0,Y 331.429,Z 329.894,A -85,B 0,C 180,E1 -14821.85,E2 -14821.85} C_VEL
LIN {X 0,Y 332.489,Z 336.276,A -85,B 0,C 180,E1 -14823.65,E2 -14823.65} C_VEL
LIN {X 0,Y 332.358,Z 337.531,A -85,B 0,C 180,E1 -14823.968,E2 -14823.968} C_VEL
LIN {X 0,Y 338.036,Z 364.395,A -85,B 0,C 180,E1 -14825.184,E2 -14825.184} C_VEL
LIN {X 0,Y 340.363,Z 379.852,A -85,B 0,C 180,E1 -14825.768,E2 -14825.768} C_VEL
LIN {X 0,Y 338.595,Z 446.356,A -85,B 0,C 180,E1 -14827.22,E2 -14827.22} C_VEL
LIN {X 0,Y 337.719,Z 459.473,A -85,B 0,C 180,E1 -14827.722,E2 -14827.722} C_VEL
LIN {X 0,Y 336.396,Z 472.681,A -85,B 0,C 180,E1 -14828.477,E2 -14828.477} C_VEL
LIN {X 0,Y 334.922,Z 484.592,A -85,B 0,C 180,E1 -14829.424,E2 -14829.424} C_VEL
LIN {X 0,Y 333.198,Z 496.021,A -85,B 0,C 180,E1 -14830.599,E2 -14830.599} C_VEL
LIN {X 0,Y 331.607,Z 506.337,A -85,B 0,C 180,E1 -14831.945,E2 -14831.945} C_VEL
LIN {X 0,Y 329.951,Z 515.59,A -85,B 0,C 180,E1 -14833.438,E2 -14833.438} C_VEL
LIN {X 0,Y 328.68,Z 523.997,A -85,B 0,C 180,E1 -14835.134,E2 -14835.134} C_VEL
LIN {X 0,Y 327.262,Z 531.419,A -85,B 0,C 180,E1 -14836.97,E2 -14836.97} C_VEL
LIN {X 0,Y 326.283,Z 537.402,A -85,B 0,C 180,E1 -14838.824,E2 -14838.824} C_VEL
LIN {X 0,Y 325.593,Z 542.154,A -85,B 0,C 180,E1 -14840.685,E2 -14840.685} C_VEL
LIN {X 0,Y 325.156,Z 545.811,A -85,B 0,C 180,E1 -14842.551,E2 -14842.551} C_VEL
LIN {X 0,Y 324.924,Z 548.277,A -85,B 0,C 180,E1 -14844.251,E2 -14844.251} C_VEL
LIN {X 0,Y 324.901,Z 550.207,A -85,B 0,C 180,E1 -14846.281,E2 -14846.281} C_VEL
LIN {X 0,Y 324.871,Z 551.13,A -85,B 0,C 180,E1 -14848.762,E2 -14848.762} C_VEL
LIN {X 0,Y 324.949,Z 550.981,A -85,B 0,C 180,E1 -14850.002,E2 -14850.002} C_VEL
LIN {X 0,Y 324.904,Z 550.412,A -85,B 0,C 180,E1 -14851.241,E2 -14851.241} C_VEL
LIN {X 0,Y 324.944,Z 548.092,A -85,B 0,C 180,E1 -14853.722,E2 -14853.722} C_VEL
LIN {X 0,Y 325.019,Z 544.58,A -85,B 0,C 180,E1 -14855.913,E2 -14855.913} C_VEL
LIN {X 0,Y 325.23,Z 539.656,A -85,B 0,C 180,E1 -14858.076,E2 -14858.076} C_VEL
LIN {X 0,Y 325.618,Z 534.117,A -85,B 0,C 180,E1 -14859.945,E2 -14859.945} C_VEL
LIN {X 0,Y 326.22,Z 527.181,A -85,B 0,C 180,E1 -14861.812,E2 -14861.812} C_VEL
LIN {X 0,Y 327.055,Z 520.101,A -85,B 0,C 180,E1 -14863.358,E2 -14863.358} C_VEL
LIN {X 0,Y 328.02,Z 511.548,A -85,B 0,C 180,E1 -14864.9,E2 -14864.9} C_VEL
LIN {X 0,Y 329.07,Z 500.938,A -85,B 0,C 180,E1 -14866.44,E2 -14866.44} C_VEL
LIN {X 0,Y 330.08,Z 490.425,A -85,B 0,C 180,E1 -14867.664,E2 -14867.664} C_VEL
LIN {X 0,Y 331.192,Z 478.884,A -85,B 0,C 180,E1 -14868.722,E2 -14868.722} C_VEL
LIN {X 0,Y 332.175,Z 466.932,A -85,B 0,C 180,E1 -14869.547,E2 -14869.547} C_VEL
LIN {X 0,Y 333.031,Z 453.116,A -85,B 0,C 180,E1 -14870.218,E2 -14870.218} C_VEL
LIN {X 0,Y 333.482,Z 440.51,A -85,B 0,C 180,E1 -14870.592,E2 -14870.592} C_VEL
LIN {X 0,Y 334.576,Z 377.072,A -85,B 0,C 180,E1 -14871.95,E2 -14871.95} C_VEL
LIN {X 0,Y 329.311,Z 338.4,A -85,B 0,C 180,E1 -14873.132,E2 -14873.132} C_VEL
LIN {X 0,Y 330.291,Z 328.59,A -85,B 0,C 180,E1 -14875.525,E2 -14875.525} C_VEL
LIN {X 0,Y 328.588,Z 318.954,A -85,B 0,C 180,E1 -14878.071,E2 -14878.071} C_VEL
LIN {X 0,Y 326.637,Z 309.801,A -85,B 0,C 180,E1 -14880.61,E2 -14880.61} C_VEL
LIN {X 0,Y 326.613,Z 309.8,A -85,B 0,C 180,E1 -14884.02,E2 -14884.02} C_VEL
LIN {X 0,Y 326.634,Z 309.795,A -85,B 0,C 180,E1 -14887.239,E2 -14887.239} C_VEL
LIN {X 0,Y 326.584,Z 309.802,A -85,B 0,C 180,E1 -14891.132,E2 -14891.132} C_VEL
LIN {X 0,Y 326.534,Z 309.812,A -85,B 0,C 180,E1 -14894.743,E2 -14894.743} C_VEL
LIN {X 0,Y 326.583,Z 309.802,A -85,B 0,C 180,E1 -14898.155,E2 -14898.155} C_VEL
LIN {X 0,Y 326.604,Z 309.799,A -85,B 0,C 180,E1 -14901.388,E2 -14901.388} C_VEL
LIN {X 0,Y 326.626,Z 309.8,A -85,B 0,C 180,E1 -14904.852,E2 -14904.852} C_VEL
LIN {X 0,Y 326.614,Z 309.799,A -85,B 0,C 180,E1 -14907.456,E2 -14907.456} C_VEL
LIN {X 0,Y 326.668,Z 309.79,A -85,B 0,C 180,E1 -14910.341,E2 -14910.341} C_VEL
LIN {X 0,Y 326.697,Z 309.787,A -85,B 0,C 180,E1 -14914.517,E2 -14914.517} C_VEL
LIN {X 0,Y 326.625,Z 309.795,A -85,B 0,C 180,E1 -14918.544,E2 -14918.544} C_VEL
LIN {X 0,Y 326.67,Z 309.788,A -85,B 0,C 180,E1 -14922.47,E2 -14922.47} C_VEL
LIN {X 0,Y 326.766,Z 309.779,A -85,B 0,C 180,E1 -14926.315,E2 -14926.315} C_VEL
LIN {X 0,Y 326.811,Z 309.774,A -85,B 0,C 180,E1 -14930.093,E2 -14930.093} C_VEL
LIN {X 0,Y 326.952,Z 309.757,A -85,B 0,C 180,E1 -14933.83,E2 -14933.83} C_VEL
LIN {X 0,Y 327.051,Z 309.743,A -85,B 0,C 180,E1 -14937.537,E2 -14937.537} C_VEL
LIN {X 0,Y 327.184,Z 309.731,A -85,B 0,C 180,E1 -14940,E2 -14940} C_VEL
LIN {X 0,Y 327.051,Z 309.744,A -85,B 0,C 180,E1 -14942.463,E2 -14942.463} C_VEL
LIN {X 0,Y 326.956,Z 309.752,A -85,B 0,C 180,E1 -14946.599,E2 -14946.599} C_VEL
LIN {X 0,Y 326.789,Z 309.776,A -85,B 0,C 180,E1 -14949.907,E2 -14949.907} C_VEL
LIN {X 0,Y 326.765,Z 309.778,A -85,B 0,C 180,E1 -14953.685,E2 -14953.685} C_VEL
LIN {X 0,Y 326.67,Z 309.79,A -85,B 0,C 180,E1 -14957.529,E2 -14957.529} C_VEL
LIN {X 0,Y 326.624,Z 309.796,A -85,B 0,C 180,E1 -14961.456,E2 -14961.456} C_VEL
LIN {X 0,Y 326.696,Z 309.788,A -85,B 0,C 180,E1 -14965.483,E2 -14965.483} C_VEL
LIN {X 0,Y 326.653,Z 309.792,A -85,B 0,C 180,E1 -14969.66,E2 -14969.66} C_VEL
LIN {X 0,Y 326.612,Z 309.796,A -85,B 0,C 180,E1 -14974.019,E2 -14974.019} C_VEL
LIN {X 0,Y 326.632,Z 309.799,A -85,B 0,C 180,E1 -14977.238,E2 -14977.238} C_VEL
LIN {X 0,Y 326.583,Z 309.802,A -85,B 0,C 180,E1 -14981.13,E2 -14981.13} C_VEL
LIN {X 0,Y 326.532,Z 309.807,A -85,B 0,C 180,E1 -14984.742,E2 -14984.742} C_VEL
LIN {X 0,Y 326.58,Z 309.803,A -85,B 0,C 180,E1 -14988.153,E2 -14988.153} C_VEL
LIN {X 0,Y 326.627,Z 309.797,A -85,B 0,C 180,E1 -14991.39,E2 -14991.39} C_VEL
LIN {X 0,Y 326.623,Z 309.795,A -85,B 0,C 180,E1 -14994.85,E2 -14994.85} C_VEL
LIN {X 0,Y 326.612,Z 309.799,A -85,B 0,C 180,E1 -14997.454,E2 -14997.454} C_VEL
LIN {X 0,Y 326.651,Z 309.796,A -85,B 0,C 180,E1 -15000.338,E2 -15000.338} C_VEL
LIN {X 0,Y 326.693,Z 309.79,A -85,B 0,C 180,E1 -15004.515,E2 -15004.515} C_VEL
LIN {X 0,Y 326.656,Z 309.796,A -85,B 0,C 180,E1 -15008.544,E2 -15008.544} C_VEL
LIN {X 0,Y 326.747,Z 309.781,A -85,B 0,C 180,E1 -15011.176,E2 -15011.176} C_VEL
LIN {X 0,Y 326.765,Z 309.779,A -85,B 0,C 180,E1 -15015.431,E2 -15015.431} C_VEL
LIN {X 0,Y 326.76,Z 309.784,A -85,B 0,C 180,E1 -15018.837,E2 -15018.837} C_VEL
LIN {X 0,Y 326.789,Z 309.861,A -85,B 0,C 180,E1 -15020.131,E2 -15020.131} C_VEL
LIN {X 0,Y 328.059,Z 315.738,A -85,B 0,C 180,E1 -15021.854,E2 -15021.854} C_VEL
LIN {X 0,Y 332.563,Z 330.036,A -85,B 0,C 180,E1 -15022.474,E2 -15022.474} C_VEL
LIN {X 0,Y 335.132,Z 344.32,A -85,B 0,C 180,E1 -15022.944,E2 -15022.944} C_VEL
LIN {X 0,Y 333.48,Z 423.822,A -85,B 0,C 180,E1 -15024.67,E2 -15024.67} C_VEL
LIN {X 0,Y 332.876,Z 437.56,A -85,B 0,C 180,E1 -15025.23,E2 -15025.23} C_VEL
LIN {X 0,Y 332.201,Z 449.877,A -85,B 0,C 180,E1 -15025.98,E2 -15025.98} C_VEL
LIN {X 0,Y 331.352,Z 461.474,A -85,B 0,C 180,E1 -15026.935,E2 -15026.935} C_VEL
LIN {X 0,Y 330.281,Z 472.612,A -85,B 0,C 180,E1 -15028.108,E2 -15028.108} C_VEL
LIN {X 0,Y 329.114,Z 483.423,A -85,B 0,C 180,E1 -15029.539,E2 -15029.539} C_VEL
LIN {X 0,Y 327.984,Z 493.47,A -85,B 0,C 180,E1 -15031.226,E2 -15031.226} C_VEL
LIN {X 0,Y 326.974,Z 502.312,A -85,B 0,C 180,E1 -15033.078,E2 -15033.078} C_VEL
LIN {X 0,Y 326.198,Z 509.377,A -85,B 0,C 180,E1 -15034.942,E2 -15034.942} C_VEL
LIN {X 0,Y 325.729,Z 515.546,A -85,B 0,C 180,E1 -15037.021,E2 -15037.021} C_VEL
LIN {X 0,Y 325.209,Z 520.709,A -85,B 0,C 180,E1 -15039.326,E2 -15039.326} C_VEL
LIN {X 0,Y 324.921,Z 523.725,A -85,B 0,C 180,E1 -15041.223,E2 -15041.223} C_VEL
LIN {X 0,Y 324.821,Z 525.789,A -85,B 0,C 180,E1 -15043.185,E2 -15043.185} C_VEL
LIN {X 0,Y 324.717,Z 526.808,A -85,B 0,C 180,E1 -15045.051,E2 -15045.051} C_VEL
LIN {X 0,Y 324.75,Z 527.002,A -85,B 0,C 180,E1 -15046.338,E2 -15046.338} C_VEL
LIN {X 0,Y 324.898,Z 526.662,A -85,B 0,C 180,E1 -15047.866,E2 -15047.866} C_VEL
LIN {X 0,Y 325.226,Z 525.014,A -85,B 0,C 180,E1 -15050.226,E2 -15050.226} C_VEL
LIN {X 0,Y 325.656,Z 522.945,A -85,B 0,C 180,E1 -15051.878,E2 -15051.878} C_VEL
LIN {X 0,Y 326.387,Z 518.903,A -85,B 0,C 180,E1 -15054.147,E2 -15054.147} C_VEL
LIN {X 0,Y 327.291,Z 514.062,A -85,B 0,C 180,E1 -15056.114,E2 -15056.114} C_VEL
LIN {X 0,Y 328.471,Z 507.826,A -85,B 0,C 180,E1 -15058.078,E2 -15058.078} C_VEL
LIN {X 0,Y 329.985,Z 499.964,A -85,B 0,C 180,E1 -15060.031,E2 -15060.031} C_VEL
LIN {X 0,Y 331.478,Z 491.809,A -85,B 0,C 180,E1 -15061.649,E2 -15061.649} C_VEL
LIN {X 0,Y 333.067,Z 481.665,A -85,B 0,C 180,E1 -15063.27,E2 -15063.27} C_VEL
LIN {X 0,Y 334.668,Z 471.687,A -85,B 0,C 180,E1 -15064.538,E2 -15064.538} C_VEL
LIN {X 0,Y 336.179,Z 460.094,A -85,B 0,C 180,E1 -15065.715,E2 -15065.715} C_VEL
LIN {X 0,Y 337.412,Z 447.473,A -85,B 0,C 180,E1 -15066.691,E2 -15066.691} C_VEL
LIN {X 0,Y 338.512,Z 434.458,A -85,B 0,C 180,E1 -15067.408,E2 -15067.408} C_VEL
LIN {X 0,Y 339.157,Z 421.304,A -85,B 0,C 180,E1 -15067.873,E2 -15067.873} C_VEL
LIN {X 0,Y 340.604,Z 368.554,A -85,B 0,C 180,E1 -15069.013,E2 -15069.013} C_VEL
LIN {X 0,Y 340.255,Z 362.712,A -85,B 0,C 180,E1 -15069.185,E2 -15069.185} C_VEL
LIN {X 0,Y 338.992,Z 357.074,A -85,B 0,C 180,E1 -15069.437,E2 -15069.437} C_VEL
LIN {X 0,Y 337.796,Z 353.455,A -85,B 0,C 180,E1 -15069.637,E2 -15069.637} C_VEL
LIN {X 0,Y 331.784,Z 339.353,A -85,B 0,C 180,E1 -15070.571,E2 -15070.571} C_VEL
LIN {X 0,Y 324.512,Z 323.612,A -85,B 0,C 180,E1 -15071.732,E2 -15071.732} C_VEL
LIN {X 0,Y 321.093,Z 316.717,A -85,B 0,C 180,E1 -15072.299,E2 -15072.299} C_VEL
LIN {X 0,Y 319.508,Z 310.686,A -85,B 0,C 180,E1 -15074.387,E2 -15074.387} C_VEL
LIN {X 0,Y 319.54,Z 310.675,A -85,B 0,C 180,E1 -15077.015,E2 -15077.015} C_VEL
LIN {X 0,Y 319.503,Z 310.688,A -85,B 0,C 180,E1 -15080.365,E2 -15080.365} C_VEL
LIN {X 0,Y 319.565,Z 310.659,A -85,B 0,C 180,E1 -15084.457,E2 -15084.457} C_VEL
LIN {X 0,Y 319.511,Z 310.681,A -85,B 0,C 180,E1 -15088.136,E2 -15088.136} C_VEL
LIN {X 0,Y 319.558,Z 310.675,A -85,B 0,C 180,E1 -15091.603,E2 -15091.603} C_VEL
LIN {X 0,Y 319.56,Z 310.672,A -85,B 0,C 180,E1 -15095.301,E2 -15095.301} C_VEL
LIN {X 0,Y 319.589,Z 310.666,A -85,B 0,C 180,E1 -15099.4,E2 -15099.4} C_VEL
LIN {X 0,Y 319.644,Z 310.665,A -85,B 0,C 180,E1 -15102.073,E2 -15102.073} C_VEL
LIN {X 0,Y 319.718,Z 310.661,A -85,B 0,C 180,E1 -15106.007,E2 -15106.007} C_VEL
LIN {X 0,Y 319.738,Z 310.655,A -85,B 0,C 180,E1 -15109.873,E2 -15109.873} C_VEL
LIN {X 0,Y 319.894,Z 310.626,A -85,B 0,C 180,E1 -15113.694,E2 -15113.694} C_VEL
LIN {X 0,Y 319.975,Z 310.618,A -85,B 0,C 180,E1 -15117.483,E2 -15117.483} C_VEL
LIN {X 0,Y 320.136,Z 310.603,A -85,B 0,C 180,E1 -15120,E2 -15120} C_VEL
LIN {X 0,Y 319.975,Z 310.616,A -85,B 0,C 180,E1 -15122.518,E2 -15122.518} C_VEL
LIN {X 0,Y 319.937,Z 310.632,A -85,B 0,C 180,E1 -15126.306,E2 -15126.306} C_VEL
LIN {X 0,Y 319.829,Z 310.633,A -85,B 0,C 180,E1 -15128.849,E2 -15128.849} C_VEL
LIN {X 0,Y 319.669,Z 310.657,A -85,B 0,C 180,E1 -15132.701,E2 -15132.701} C_VEL
LIN {X 0,Y 319.687,Z 310.661,A -85,B 0,C 180,E1 -15135.296,E2 -15135.296} C_VEL
LIN {X 0,Y 319.663,Z 310.657,A -85,B 0,C 180,E1 -15139.256,E2 -15139.256} C_VEL
LIN {X 0,Y 319.558,Z 310.669,A -85,B 0,C 180,E1 -15143.321,E2 -15143.321} C_VEL
LIN {X 0,Y 319.624,Z 310.67,A -85,B 0,C 180,E1 -15146.089,E2 -15146.089} C_VEL
LIN {X 0,Y 319.579,Z 310.67,A -85,B 0,C 180,E1 -15148.935,E2 -15148.935} C_VEL
LIN {X 0,Y 319.528,Z 310.675,A -85,B 0,C 180,E1 -15151.863,E2 -15151.863} C_VEL
LIN {X 0,Y 319.571,Z 310.674,A -85,B 0,C 180,E1 -15155.545,E2 -15155.545} C_VEL
LIN {X 0,Y 319.589,Z 310.677,A -85,B 0,C 180,E1 -15158.006,E2 -15158.006} C_VEL
LIN {X 0,Y 319.564,Z 310.678,A -85,B 0,C 180,E1 -15161.608,E2 -15161.608} C_VEL
LIN {X 0,Y 319.57,Z 310.665,A -85,B 0,C 180,E1 -15165.275,E2 -15165.275} C_VEL
LIN {X 0,Y 319.576,Z 310.677,A -85,B 0,C 180,E1 -15168.722,E2 -15168.722} C_VEL
LIN {X 0,Y 319.592,Z 310.677,A -85,B 0,C 180,E1 -15172.341,E2 -15172.341} C_VEL
LIN {X 0,Y 319.603,Z 310.815,A -85,B 0,C 180,E1 -15175.048,E2 -15175.048} C_VEL
LIN {X 0,Y 322.24,Z 321.174,A -85,B 0,C 180,E1 -15178.44,E2 -15178.44} C_VEL
LIN {X 0,Y 324.533,Z 331.338,A -85,B 0,C 180,E1 -15181.55,E2 -15181.55} C_VEL
LIN {X 0,Y 325.622,Z 337.238,A -85,B 0,C 180,E1 -15183.267,E2 -15183.267} C_VEL
LIN {X 0,Y 328.777,Z 350.638,A -85,B 0,C 180,E1 -15183.94,E2 -15183.94} C_VEL
LIN {X 0,Y 332.501,Z 369.494,A -85,B 0,C 180,E1 -15184.781,E2 -15184.781} C_VEL
LIN {X 0,Y 334.099,Z 380.253,A -85,B 0,C 180,E1 -15185.197,E2 -15185.197} C_VEL
LIN {X 0,Y 332.269,Z 446.595,A -85,B 0,C 180,E1 -15186.678,E2 -15186.678} C_VEL
LIN {X 0,Y 331.294,Z 460.298,A -85,B 0,C 180,E1 -15187.225,E2 -15187.225} C_VEL
LIN {X 0,Y 329.958,Z 472.662,A -85,B 0,C 180,E1 -15187.953,E2 -15187.953} C_VEL
LIN {X 0,Y 328.531,Z 483.719,A -85,B 0,C 180,E1 -15188.841,E2 -15188.841} C_VEL
LIN {X 0,Y 326.78,Z 495.245,A -85,B 0,C 180,E1 -15190.039,E2 -15190.039} C_VEL
LIN {X 0,Y 325.048,Z 505.642,A -85,B 0,C 180,E1 -15191.405,E2 -15191.405} C_VEL
LIN {X 0,Y 323.293,Z 514.924,A -85,B 0,C 180,E1 -15192.913,E2 -15192.913} C_VEL
LIN {X 0,Y 321.812,Z 524.119,A -85,B 0,C 180,E1 -15194.809,E2 -15194.809} C_VEL
LIN {X 0,Y 320.352,Z 531.471,A -85,B 0,C 180,E1 -15196.684,E2 -15196.684} C_VEL
LIN {X 0,Y 319.275,Z 537.393,A -85,B 0,C 180,E1 -15198.576,E2 -15198.576} C_VEL
LIN {X 0,Y 318.576,Z 542.091,A -85,B 0,C 180,E1 -15200.478,E2 -15200.478} C_VEL
LIN {X 0,Y 318.084,Z 545.696,A -85,B 0,C 180,E1 -15202.384,E2 -15202.384} C_VEL
LIN {X 0,Y 317.843,Z 548.3,A -85,B 0,C 180,E1 -15204.282,E2 -15204.282} C_VEL
LIN {X 0,Y 317.809,Z 549.998,A -85,B 0,C 180,E1 -15206.198,E2 -15206.198} C_VEL
LIN {X 0,Y 317.778,Z 550.63,A -85,B 0,C 180,E1 -15207.467,E2 -15207.467} C_VEL
LIN {X 0,Y 317.78,Z 550.871,A -85,B 0,C 180,E1 -15208.735,E2 -15208.735} C_VEL
LIN {X 0,Y 317.854,Z 550.681,A -85,B 0,C 180,E1 -15210.002,E2 -15210.002} C_VEL
LIN {X 0,Y 317.812,Z 550.089,A -85,B 0,C 180,E1 -15211.269,E2 -15211.269} C_VEL
LIN {X 0,Y 317.801,Z 549.105,A -85,B 0,C 180,E1 -15212.537,E2 -15212.537} C_VEL
LIN {X 0,Y 317.85,Z 547.717,A -85,B 0,C 180,E1 -15213.805,E2 -15213.805} C_VEL
LIN {X 0,Y 317.914,Z 544.532,A -85,B 0,C 180,E1 -15215.843,E2 -15215.843} C_VEL
LIN {X 0,Y 318.064,Z 540.767,A -85,B 0,C 180,E1 -15217.62,E2 -15217.62} C_VEL
LIN {X 0,Y 318.505,Z 534.58,A -85,B 0,C 180,E1 -15219.848,E2 -15219.848} C_VEL
LIN {X 0,Y 319.113,Z 527.807,A -85,B 0,C 180,E1 -15221.756,E2 -15221.756} C_VEL
LIN {X 0,Y 320.071,Z 519.395,A -85,B 0,C 180,E1 -15223.655,E2 -15223.655} C_VEL
LIN {X 0,Y 321.067,Z 510.714,A -85,B 0,C 180,E1 -15225.231,E2 -15225.231} C_VEL
LIN {X 0,Y 322.211,Z 499.986,A -85,B 0,C 180,E1 -15226.8,E2 -15226.8} C_VEL
LIN {X 0,Y 323.116,Z 490.766,A -85,B 0,C 180,E1 -15227.894,E2 -15227.894} C_VEL
LIN {X 0,Y 324.246,Z 479.378,A -85,B 0,C 180,E1 -15228.975,E2 -15228.975} C_VEL
LIN {X 0,Y 325.253,Z 467.761,A -85,B 0,C 180,E1 -15229.816,E2 -15229.816} C_VEL
LIN {X 0,Y 326.133,Z 454.393,A -85,B 0,C 180,E1 -15230.5,E2 -15230.5} C_VEL
LIN {X 0,Y 326.648,Z 441.348,A -85,B 0,C 180,E1 -15230.919,E2 -15230.919} C_VEL
LIN {X 0,Y 327.785,Z 377.674,A -85,B 0,C 180,E1 -15232.313,E2 -15232.313} C_VEL
LIN {X 0,Y 322.445,Z 338.164,A -85,B 0,C 180,E1 -15233.542,E2 -15233.542} C_VEL
LIN {X 0,Y 323.268,Z 329.236,A -85,B 0,C 180,E1 -15235.775,E2 -15235.775} C_VEL
LIN {X 0,Y 321.125,Z 317.732,A -85,B 0,C 180,E1 -15238.904,E2 -15238.904} C_VEL
LIN {X 0,Y 319.578,Z 310.681,A -85,B 0,C 180,E1 -15240.944,E2 -15240.944} C_VEL
LIN {X 0,Y 319.566,Z 310.677,A -85,B 0,C 180,E1 -15244.878,E2 -15244.878} C_VEL
LIN {X 0,Y 319.563,Z 310.678,A -85,B 0,C 180,E1 -15248.011,E2 -15248.011} C_VEL
LIN {X 0,Y 319.532,Z 310.68,A -85,B 0,C 180,E1 -15251.598,E2 -15251.598} C_VEL
LIN {X 0,Y 319.495,Z 310.685,A -85,B 0,C 180,E1 -15255.258,E2 -15255.258} C_VEL
LIN {X 0,Y 319.536,Z 310.685,A -85,B 0,C 180,E1 -15258.713,E2 -15258.713} C_VEL
LIN {X 0,Y 319.56,Z 310.677,A -85,B 0,C 180,E1 -15262.35,E2 -15262.35} C_VEL
LIN {X 0,Y 319.567,Z 310.678,A -85,B 0,C 180,E1 -15265.124,E2 -15265.124} C_VEL
LIN {X 0,Y 319.577,Z 310.679,A -85,B 0,C 180,E1 -15269.058,E2 -15269.058} C_VEL
LIN {X 0,Y 319.615,Z 310.669,A -85,B 0,C 180,E1 -15272.498,E2 -15272.498} C_VEL
LIN {X 0,Y 319.611,Z 310.675,A -85,B 0,C 180,E1 -15275.304,E2 -15275.304} C_VEL
LIN {X 0,Y 319.589,Z 310.677,A -85,B 0,C 180,E1 -15279.399,E2 -15279.399} C_VEL
LIN {X 0,Y 319.658,Z 310.665,A -85,B 0,C 180,E1 -15283.392,E2 -15283.392} C_VEL
LIN {X 0,Y 319.739,Z 310.656,A -85,B 0,C 180,E1 -15286.008,E2 -15286.008} C_VEL
LIN {X 0,Y 319.758,Z 310.654,A -85,B 0,C 180,E1 -15289.873,E2 -15289.873} C_VEL
LIN {X 0,Y 319.909,Z 310.632,A -85,B 0,C 180,E1 -15293.693,E2 -15293.693} C_VEL
LIN {X 0,Y 319.995,Z 310.622,A -85,B 0,C 180,E1 -15297.482,E2 -15297.482} C_VEL
LIN {X 0,Y 320.136,Z 310.609,A -85,B 0,C 180,E1 -15300,E2 -15300} C_VEL
LIN {X 0,Y 319.994,Z 310.622,A -85,B 0,C 180,E1 -15302.517,E2 -15302.517} C_VEL
LIN {X 0,Y 319.919,Z 310.629,A -85,B 0,C 180,E1 -15306.585,E2 -15306.585} C_VEL
LIN {X 0,Y 319.742,Z 310.655,A -85,B 0,C 180,E1 -15310.127,E2 -15310.127} C_VEL
LIN {X 0,Y 319.739,Z 310.654,A -85,B 0,C 180,E1 -15313.992,E2 -15313.992} C_VEL
LIN {X 0,Y 319.62,Z 310.668,A -85,B 0,C 180,E1 -15317.929,E2 -15317.929} C_VEL
LIN {X 0,Y 319.574,Z 310.673,A -85,B 0,C 180,E1 -15321.954,E2 -15321.954} C_VEL
LIN {X 0,Y 319.624,Z 310.668,A -85,B 0,C 180,E1 -15326.089,E2 -15326.089} C_VEL
LIN {X 0,Y 319.586,Z 310.676,A -85,B 0,C 180,E1 -15328.934,E2 -15328.934} C_VEL
LIN {X 0,Y 319.536,Z 310.679,A -85,B 0,C 180,E1 -15331.861,E2 -15331.861} C_VEL
LIN {X 0,Y 319.585,Z 310.675,A -85,B 0,C 180,E1 -15335.542,E2 -15335.542} C_VEL
LIN {X 0,Y 319.564,Z 310.677,A -85,B 0,C 180,E1 -15339.668,E2 -15339.668} C_VEL
LIN {X 0,Y 319.526,Z 310.685,A -85,B 0,C 180,E1 -15343.459,E2 -15343.459} C_VEL
LIN {X 0,Y 319.559,Z 310.676,A -85,B 0,C 180,E1 -15347.015,E2 -15347.015} C_VEL
LIN {X 0,Y 319.551,Z 310.677,A -85,B 0,C 180,E1 -15350.37,E2 -15350.37} C_VEL
LIN {X 0,Y 319.562,Z 310.679,A -85,B 0,C 180,E1 -15353.571,E2 -15353.571} C_VEL
LIN {X 0,Y 319.581,Z 310.674,A -85,B 0,C 180,E1 -15356.685,E2 -15356.685} C_VEL
LIN {X 0,Y 319.588,Z 310.674,A -85,B 0,C 180,E1 -15359.615,E2 -15359.615} C_VEL
LIN {X 0,Y 319.609,Z 310.672,A -85,B 0,C 180,E1 -15362.496,E2 -15362.496} C_VEL
LIN {X 0,Y 319.608,Z 310.67,A -85,B 0,C 180,E1 -15365.303,E2 -15365.303} C_VEL
LIN {X 0,Y 319.625,Z 310.667,A -85,B 0,C 180,E1 -15369.4,E2 -15369.4} C_VEL
LIN {X 0,Y 319.662,Z 310.666,A -85,B 0,C 180,E1 -15372.072,E2 -15372.072} C_VEL
LIN {X 0,Y 319.734,Z 310.656,A -85,B 0,C 180,E1 -15376.006,E2 -15376.006} C_VEL
LIN {X 0,Y 319.755,Z 310.742,A -85,B 0,C 180,E1 -15379.831,E2 -15379.831} C_VEL
LIN {X 0,Y 320.919,Z 316.081,A -85,B 0,C 180,E1 -15381.437,E2 -15381.437} C_VEL
LIN {X 0,Y 326.068,Z 332.255,A -85,B 0,C 180,E1 -15382.14,E2 -15382.14} C_VEL
LIN {X 0,Y 328.298,Z 343.973,A -85,B 0,C 180,E1 -15382.541,E2 -15382.541} C_VEL
LIN {X 0,Y 326.673,Z 424.242,A -85,B 0,C 180,E1 -15384.326,E2 -15384.326} C_VEL
LIN {X 0,Y 326.046,Z 437.929,A -85,B 0,C 180,E1 -15384.897,E2 -15384.897} C_VEL
LIN {X 0,Y 325.351,Z 450.209,A -85,B 0,C 180,E1 -15385.662,E2 -15385.662} C_VEL
LIN {X 0,Y 324.438,Z 462.18,A -85,B 0,C 180,E1 -15386.675,E2 -15386.675} C_VEL
LIN {X 0,Y 323.273,Z 474.069,A -85,B 0,C 180,E1 -15387.973,E2 -15387.973} C_VEL
LIN {X 0,Y 322.122,Z 484.214,A -85,B 0,C 180,E1 -15389.373,E2 -15389.373} C_VEL
LIN {X 0,Y 321.04,Z 493.352,A -85,B 0,C 180,E1 -15390.939,E2 -15390.939} C_VEL
LIN {X 0,Y 319.987,Z 502.258,A -85,B 0,C 180,E1 -15392.831,E2 -15392.831} C_VEL
LIN {X 0,Y 319.205,Z 509.399,A -85,B 0,C 180,E1 -15394.734,E2 -15394.734} C_VEL
LIN {X 0,Y 318.824,Z 514.217,A -85,B 0,C 180,E1 -15396.326,E2 -15396.326} C_VEL
LIN {X 0,Y 318.333,Z 518.911,A -85,B 0,C 180,E1 -15398.249,E2 -15398.249} C_VEL
LIN {X 0,Y 317.963,Z 522.489,A -85,B 0,C 180,E1 -15400.183,E2 -15400.183} C_VEL
LIN {X 0,Y 317.814,Z 524.286,A -85,B 0,C 180,E1 -15401.478,E2 -15401.478} C_VEL
LIN {X 0,Y 317.737,Z 526.095,A -85,B 0,C 180,E1 -15403.287,E2 -15403.287} C_VEL
LIN {X 0,Y 317.639,Z 527.151,A -85,B 0,C 180,E1 -15405.395,E2 -15405.395} C_VEL
LIN {X 0,Y 317.696,Z 527.24,A -85,B 0,C 180,E1 -15406.711,E2 -15406.711} C_VEL
LIN {X 0,Y 317.838,Z 526.92,A -85,B 0,C 180,E1 -15408.046,E2 -15408.046} C_VEL
LIN {X 0,Y 317.984,Z 526.202,A -85,B 0,C 180,E1 -15409.359,E2 -15409.359} C_VEL
LIN {X 0,Y 318.245,Z 524.998,A -85,B 0,C 180,E1 -15410.689,E2 -15410.689} C_VEL
LIN {X 0,Y 318.632,Z 523.213,A -85,B 0,C 180,E1 -15412.123,E2 -15412.123} C_VEL
LIN {X 0,Y 319.273,Z 519.981,A -85,B 0,C 180,E1 -15414.029,E2 -15414.029} C_VEL
LIN {X 0,Y 320.175,Z 515.42,A -85,B 0,C 180,E1 -15416.038,E2 -15416.038} C_VEL
LIN {X 0,Y 321.38,Z 509.526,A -85,B 0,C 180,E1 -15418.043,E2 -15418.043} C_VEL
LIN {X 0,Y 322.911,Z 501.993,A -85,B 0,C 180,E1 -15420.036,E2 -15420.036} C_VEL
LIN {X 0,Y 324.376,Z 494.245,A -85,B 0,C 180,E1 -15421.688,E2 -15421.688} C_VEL
LIN {X 0,Y 326.077,Z 484.7,A -85,B 0,C 180,E1 -15423.337,E2 -15423.337} C_VEL
LIN {X 0,Y 327.873,Z 473.995,A -85,B 0,C 180,E1 -15424.797,E2 -15424.797} C_VEL
LIN {X 0,Y 329.463,Z 462.551,A -85,B 0,C 180,E1 -15426.032,E2 -15426.032} C_VEL
LIN {X 0,Y 330.844,Z 450.139,A -85,B 0,C 180,E1 -15427.065,E2 -15427.065} C_VEL
LIN {X 0,Y 331.967,Z 437.435,A -85,B 0,C 180,E1 -15427.825,E2 -15427.825} C_VEL
LIN {X 0,Y 332.758,Z 423.843,A -85,B 0,C 180,E1 -15428.371,E2 -15428.371} C_VEL
LIN {X 0,Y 334.856,Z 347.834,A -85,B 0,C 180,E1 -15430.056,E2 -15430.056} C_VEL
LIN {X 0,Y 333.793,Z 344.196,A -85,B 0,C 180,E1 -15430.249,E2 -15430.249} C_VEL
LIN {X 0,Y 331.784,Z 339.353,A -85,B 0,C 180,E1 -15430.571,E2 -15430.571} C_VEL
LIN {X 0,Y 328.999,Z 334.679,A -85,B 0,C 180,E1 -15430.973,E2 -15430.973} C_VEL
LIN {X 0,Y 322.859,Z 328.338,A -85,B 0,C 180,E1 -15431.789,E2 -15431.789} C_VEL
LIN {X 0,Y 316.765,Z 322.013,A -85,B 0,C 180,E1 -15432.639,E2 -15432.639} C_VEL
LIN {X 0,Y 314.036,Z 317.362,A -85,B 0,C 180,E1 -15433.084,E2 -15433.084} C_VEL
LIN {X 0,Y 313.449,Z 315.399,A -85,B 0,C 180,E1 -15433.691,E2 -15433.691} C_VEL
LIN {X 0,Y 312.454,Z 311.562,A -85,B 0,C 180,E1 -15435.113,E2 -15435.113} C_VEL
LIN {X 0,Y 312.444,Z 311.568,A -85,B 0,C 180,E1 -15437.923,E2 -15437.923} C_VEL
LIN {X 0,Y 312.464,Z 311.568,A -85,B 0,C 180,E1 -15441.923,E2 -15441.923} C_VEL
LIN {X 0,Y 312.517,Z 311.537,A -85,B 0,C 180,E1 -15444.219,E2 -15444.219} C_VEL
LIN {X 0,Y 312.489,Z 311.563,A -85,B 0,C 180,E1 -15447.332,E2 -15447.332} C_VEL
LIN {X 0,Y 312.493,Z 311.556,A -85,B 0,C 180,E1 -15451.291,E2 -15451.291} C_VEL
LIN {X 0,Y 312.534,Z 311.549,A -85,B 0,C 180,E1 -15454.707,E2 -15454.707} C_VEL
LIN {X 0,Y 312.55,Z 311.554,A -85,B 0,C 180,E1 -15457.526,E2 -15457.526} C_VEL
LIN {X 0,Y 312.625,Z 311.544,A -85,B 0,C 180,E1 -15461.656,E2 -15461.656} C_VEL
LIN {X 0,Y 312.68,Z 311.536,A -85,B 0,C 180,E1 -15465.686,E2 -15465.686} C_VEL
LIN {X 0,Y 312.684,Z 311.532,A -85,B 0,C 180,E1 -15469.642,E2 -15469.642} C_VEL
LIN {X 0,Y 312.788,Z 311.513,A -85,B 0,C 180,E1 -15472.252,E2 -15472.252} C_VEL
LIN {X 0,Y 312.692,Z 311.534,A -85,B 0,C 180,E1 -15474.842,E2 -15474.842} C_VEL
LIN {X 0,Y 312.976,Z 311.488,A -85,B 0,C 180,E1 -15478.714,E2 -15478.714} C_VEL
LIN {X 0,Y 312.979,Z 311.495,A -85,B 0,C 180,E1 -15481.287,E2 -15481.287} C_VEL
LIN {X 0,Y 312.703,Z 311.531,A -85,B 0,C 180,E1 -15485.158,E2 -15485.158} C_VEL
LIN {X 0,Y 312.859,Z 311.505,A -85,B 0,C 180,E1 -15487.746,E2 -15487.746} C_VEL
LIN {X 0,Y 312.656,Z 311.536,A -85,B 0,C 180,E1 -15491.672,E2 -15491.672} C_VEL
LIN {X 0,Y 312.687,Z 311.527,A -85,B 0,C 180,E1 -15494.888,E2 -15494.888} C_VEL
LIN {X 0,Y 312.619,Z 311.534,A -85,B 0,C 180,E1 -15499.238,E2 -15499.238} C_VEL
LIN {X 0,Y 312.534,Z 311.547,A -85,B 0,C 180,E1 -15502.79,E2 -15502.79} C_VEL
LIN {X 0,Y 312.572,Z 311.549,A -85,B 0,C 180,E1 -15506.724,E2 -15506.724} C_VEL
LIN {X 0,Y 312.536,Z 311.556,A -85,B 0,C 180,E1 -15509.651,E2 -15509.651} C_VEL
LIN {X 0,Y 312.51,Z 311.561,A -85,B 0,C 180,E1 -15513.691,E2 -15513.691} C_VEL
LIN {X 0,Y 312.543,Z 311.557,A -85,B 0,C 180,E1 -15517.383,E2 -15517.383} C_VEL
LIN {X 0,Y 312.494,Z 311.562,A -85,B 0,C 180,E1 -15520.709,E2 -15520.709} C_VEL
LIN {X 0,Y 312.522,Z 311.554,A -85,B 0,C 180,E1 -15524.198,E2 -15524.198} C_VEL
LIN {X 0,Y 312.543,Z 311.555,A -85,B 0,C 180,E1 -15527.907,E2 -15527.907} C_VEL
LIN {X 0,Y 312.552,Z 311.557,A -85,B 0,C 180,E1 -15531.907,E2 -15531.907} C_VEL
LIN {X 0,Y 312.532,Z 311.631,A -85,B 0,C 180,E1 -15534.322,E2 -15534.322} C_VEL
LIN {X 0,Y 315.307,Z 322.138,A -85,B 0,C 180,E1 -15537.887,E2 -15537.887} C_VEL
LIN {X 0,Y 317.656,Z 332.727,A -85,B 0,C 180,E1 -15541.222,E2 -15541.222} C_VEL
LIN {X 0,Y 318.491,Z 336.966,A -85,B 0,C 180,E1 -15542.487,E2 -15542.487} C_VEL
LIN {X 0,Y 320.504,Z 342.274,A -85,B 0,C 180,E1 -15542.85,E2 -15542.85} C_VEL
LIN {X 0,Y 325.632,Z 366.685,A -85,B 0,C 180,E1 -15544.024,E2 -15544.024} C_VEL
LIN {X 0,Y 327.877,Z 381.164,A -85,B 0,C 180,E1 -15544.617,E2 -15544.617} C_VEL
LIN {X 0,Y 326.047,Z 445.708,A -85,B 0,C 180,E1 -15546.079,E2 -15546.079} C_VEL
LIN {X 0,Y 325.101,Z 458.861,A -85,B 0,C 180,E1 -15546.597,E2 -15546.597} C_VEL
LIN {X 0,Y 323.708,Z 471.536,A -85,B 0,C 180,E1 -15547.336,E2 -15547.336} C_VEL
LIN {X 0,Y 322.233,Z 482.826,A -85,B 0,C 180,E1 -15548.239,E2 -15548.239} C_VEL
LIN {X 0,Y 320.369,Z 494.481,A -85,B 0,C 180,E1 -15549.454,E2 -15549.454} C_VEL
LIN {X 0,Y 318.55,Z 504.963,A -85,B 0,C 180,E1 -15550.844,E2 -15550.844} C_VEL
LIN {X 0,Y 316.837,Z 513.56,A -85,B 0,C 180,E1 -15552.244,E2 -15552.244} C_VEL
LIN {X 0,Y 315.488,Z 521.491,A -85,B 0,C 180,E1 -15553.834,E2 -15553.834} C_VEL
LIN {X 0,Y 313.932,Z 529.306,A -85,B 0,C 180,E1 -15555.746,E2 -15555.746} C_VEL
LIN {X 0,Y 312.593,Z 535.579,A -85,B 0,C 180,E1 -15557.669,E2 -15557.669} C_VEL
LIN {X 0,Y 311.746,Z 540.597,A -85,B 0,C 180,E1 -15559.612,E2 -15559.612} C_VEL
LIN {X 0,Y 311.191,Z 544.506,A -85,B 0,C 180,E1 -15561.561,E2 -15561.561} C_VEL
LIN {X 0,Y 310.766,Z 548.316,A -85,B 0,C 180,E1 -15564.308,E2 -15564.308} C_VEL
LIN {X 0,Y 310.72,Z 549.789,A -85,B 0,C 180,E1 -15566.111,E2 -15566.111} C_VEL
LIN {X 0,Y 310.7,Z 550.399,A -85,B 0,C 180,E1 -15567.409,E2 -15567.409} C_VEL
LIN {X 0,Y 310.692,Z 550.601,A -85,B 0,C 180,E1 -15568.706,E2 -15568.706} C_VEL
LIN {X 0,Y 310.761,Z 550.38,A -85,B 0,C 180,E1 -15570.002,E2 -15570.002} C_VEL
LIN {X 0,Y 310.722,Z 549.766,A -85,B 0,C 180,E1 -15571.298,E2 -15571.298} C_VEL
LIN {X 0,Y 310.723,Z 548.76,A -85,B 0,C 180,E1 -15572.595,E2 -15572.595} C_VEL
LIN {X 0,Y 310.759,Z 547.33,A -85,B 0,C 180,E1 -15573.892,E2 -15573.892} C_VEL
LIN {X 0,Y 310.825,Z 544.418,A -85,B 0,C 180,E1 -15575.8,E2 -15575.8} C_VEL
LIN {X 0,Y 311.005,Z 540.285,A -85,B 0,C 180,E1 -15577.794,E2 -15577.794} C_VEL
LIN {X 0,Y 311.476,Z 534.022,A -85,B 0,C 180,E1 -15580.073,E2 -15580.073} C_VEL
LIN {X 0,Y 312.101,Z 527.18,A -85,B 0,C 180,E1 -15582.024,E2 -15582.024} C_VEL
LIN {X 0,Y 313.096,Z 518.667,A -85,B 0,C 180,E1 -15583.965,E2 -15583.965} C_VEL
LIN {X 0,Y 314.137,Z 509.874,A -85,B 0,C 180,E1 -15585.575,E2 -15585.575} C_VEL
LIN {X 0,Y 315.342,Z 499.031,A -85,B 0,C 180,E1 -15587.177,E2 -15587.177} C_VEL
LIN {X 0,Y 316.493,Z 488.209,A -85,B 0,C 180,E1 -15588.449,E2 -15588.449} C_VEL
LIN {X 0,Y 317.728,Z 476.055,A -85,B 0,C 180,E1 -15589.547,E2 -15589.547} C_VEL
LIN {X 0,Y 318.764,Z 463.359,A -85,B 0,C 180,E1 -15590.405,E2 -15590.405} C_VEL
LIN {X 0,Y 319.535,Z 450.973,A -85,B 0,C 180,E1 -15590.985,E2 -15590.985} C_VEL
LIN {X 0,Y 319.99,Z 435.184,A -85,B 0,C 180,E1 -15591.418,E2 -15591.418} C_VEL
LIN {X 0,Y 321.077,Z 378.787,A -85,B 0,C 180,E1 -15592.672,E2 -15592.672} C_VEL
LIN {X 0,Y 315.576,Z 337.871,A -85,B 0,C 180,E1 -15593.984,E2 -15593.984} C_VEL
LIN {X 0,Y 316.307,Z 331.224,A -85,B 0,C 180,E1 -15595.677,E2 -15595.677} C_VEL
LIN {X 0,Y 314.702,Z 321.651,A -85,B 0,C 180,E1 -15598.317,E2 -15598.317} C_VEL
LIN {X 0,Y 312.525,Z 311.558,A -85,B 0,C 180,E1 -15601.221,E2 -15601.221} C_VEL
LIN {X 0,Y 312.513,Z 311.558,A -85,B 0,C 180,E1 -15604.211,E2 -15604.211} C_VEL
LIN {X 0,Y 312.532,Z 311.552,A -85,B 0,C 180,E1 -15607.386,E2 -15607.386} C_VEL
LIN {X 0,Y 312.496,Z 311.56,A -85,B 0,C 180,E1 -15610.71,E2 -15610.71} C_VEL
LIN {X 0,Y 312.458,Z 311.563,A -85,B 0,C 180,E1 -15614.21,E2 -15614.21} C_VEL
LIN {X 0,Y 312.491,Z 311.556,A -85,B 0,C 180,E1 -15617.919,E2 -15617.919} C_VEL
LIN {X 0,Y 312.505,Z 311.558,A -85,B 0,C 180,E1 -15620.972,E2 -15620.972} C_VEL
LIN {X 0,Y 312.539,Z 311.55,A -85,B 0,C 180,E1 -15624.221,E2 -15624.221} C_VEL
LIN {X 0,Y 312.511,Z 311.556,A -85,B 0,C 180,E1 -15627.334,E2 -15627.334} C_VEL
LIN {X 0,Y 312.559,Z 311.553,A -85,B 0,C 180,E1 -15631.277,E2 -15631.277} C_VEL
LIN {X 0,Y 312.592,Z 311.545,A -85,B 0,C 180,E1 -15634.711,E2 -15634.711} C_VEL
LIN {X 0,Y 312.571,Z 311.55,A -85,B 0,C 180,E1 -15637.527,E2 -15637.527} C_VEL
LIN {X 0,Y 312.574,Z 311.546,A -85,B 0,C 180,E1 -15641.652,E2 -15641.652} C_VEL
LIN {X 0,Y 312.692,Z 311.537,A -85,B 0,C 180,E1 -15645.686,E2 -15645.686} C_VEL
LIN {X 0,Y 312.705,Z 311.534,A -85,B 0,C 180,E1 -15649.642,E2 -15649.642} C_VEL
LIN {X 0,Y 312.803,Z 311.514,A -85,B 0,C 180,E1 -15652.252,E2 -15652.252} C_VEL
LIN {X 0,Y 312.709,Z 311.526,A -85,B 0,C 180,E1 -15654.842,E2 -15654.842} C_VEL
LIN {X 0,Y 312.941,Z 311.5,A -85,B 0,C 180,E1 -15657.425,E2 -15657.425} C_VEL
LIN {X 0,Y 313.089,Z 311.486,A -85,B 0,C 180,E1 -15660,E2 -15660} C_VEL
LIN {X 0,Y 312.941,Z 311.5,A -85,B 0,C 180,E1 -15662.574,E2 -15662.574} C_VEL
LIN {X 0,Y 312.886,Z 311.506,A -85,B 0,C 180,E1 -15666.562,E2 -15666.562} C_VEL
LIN {X 0,Y 312.692,Z 311.535,A -85,B 0,C 180,E1 -15670.358,E2 -15670.358} C_VEL
LIN {X 0,Y 312.674,Z 311.535,A -85,B 0,C 180,E1 -15674.864,E2 -15674.864} C_VEL
LIN {X 0,Y 312.555,Z 311.55,A -85,B 0,C 180,E1 -15679.193,E2 -15679.193} C_VEL
LIN {X 0,Y 312.532,Z 311.555,A -85,B 0,C 180,E1 -15682.78,E2 -15682.78} C_VEL
LIN {X 0,Y 312.603,Z 311.542,A -85,B 0,C 180,E1 -15685.932,E2 -15685.932} C_VEL
LIN {X 0,Y 312.544,Z 311.55,A -85,B 0,C 180,E1 -15689.65,E2 -15689.65} C_VEL
LIN {X 0,Y 312.525,Z 311.552,A -85,B 0,C 180,E1 -15693.688,E2 -15693.688} C_VEL
LIN {X 0,Y 312.525,Z 311.557,A -85,B 0,C 180,E1 -15697.385,E2 -15697.385} C_VEL
LIN {X 0,Y 312.495,Z 311.554,A -85,B 0,C 180,E1 -15700.708,E2 -15700.708} C_VEL
LIN {X 0,Y 312.456,Z 311.56,A -85,B 0,C 180,E1 -15704.209,E2 -15704.209} C_VEL
LIN {X 0,Y 312.488,Z 311.56,A -85,B 0,C 180,E1 -15707.917,E2 -15707.917} C_VEL
LIN {X 0,Y 312.539,Z 311.555,A -85,B 0,C 180,E1 -15711.909,E2 -15711.909} C_VEL
LIN {X 0,Y 312.51,Z 311.558,A -85,B 0,C 180,E1 -15715.789,E2 -15715.789} C_VEL
LIN {X 0,Y 312.524,Z 311.552,A -85,B 0,C 180,E1 -15718.852,E2 -15718.852} C_VEL
LIN {X 0,Y 312.574,Z 311.549,A -85,B 0,C 180,E1 -15721.823,E2 -15721.823} C_VEL
LIN {X 0,Y 312.589,Z 311.546,A -85,B 0,C 180,E1 -15724.709,E2 -15724.709} C_VEL
LIN {X 0,Y 312.591,Z 311.544,A -85,B 0,C 180,E1 -15727.527,E2 -15727.527} C_VEL
LIN {X 0,Y 312.642,Z 311.538,A -85,B 0,C 180,E1 -15731.655,E2 -15731.655} C_VEL
LIN {X 0,Y 312.696,Z 311.532,A -85,B 0,C 180,E1 -15735.685,E2 -15735.685} C_VEL
LIN {X 0,Y 312.706,Z 311.606,A -85,B 0,C 180,E1 -15739.517,E2 -15739.517} C_VEL
LIN {X 0,Y 313.719,Z 316.359,A -85,B 0,C 180,E1 -15740.976,E2 -15740.976} C_VEL
LIN {X 0,Y 319.436,Z 333.674,A -85,B 0,C 180,E1 -15741.767,E2 -15741.767} C_VEL
LIN {X 0,Y 321.602,Z 345.615,A -85,B 0,C 180,E1 -15742.181,E2 -15742.181} C_VEL
LIN {X 0,Y 319.874,Z 424.546,A -85,B 0,C 180,E1 -15743.968,E2 -15743.968} C_VEL
LIN {X 0,Y 319.227,Z 438.222,A -85,B 0,C 180,E1 -15744.55,E2 -15744.55} C_VEL
LIN {X 0,Y 318.512,Z 450.495,A -85,B 0,C 180,E1 -15745.331,E2 -15745.331} C_VEL
LIN {X 0,Y 317.505,Z 463.147,A -85,B 0,C 180,E1 -15746.433,E2 -15746.433} C_VEL
LIN {X 0,Y 316.296,Z 474.998,A -85,B 0,C 180,E1 -15747.77,E2 -15747.77} C_VEL
LIN {X 0,Y 315.223,Z 484.003,A -85,B 0,C 180,E1 -15749.04,E2 -15749.04} C_VEL
LIN {X 0,Y 314.128,Z 493.222,A -85,B 0,C 180,E1 -15750.639,E2 -15750.639} C_VEL
LIN {X 0,Y 312.999,Z 502.201,A -85,B 0,C 180,E1 -15752.572,E2 -15752.572} C_VEL
LIN {X 0,Y 312.199,Z 509.414,A -85,B 0,C 180,E1 -15754.517,E2 -15754.517} C_VEL
LIN {X 0,Y 311.699,Z 515.147,A -85,B 0,C 180,E1 -15756.471,E2 -15756.471} C_VEL
LIN {X 0,Y 311.202,Z 519.683,A -85,B 0,C 180,E1 -15758.439,E2 -15758.439} C_VEL
LIN {X 0,Y 310.826,Z 523.129,A -85,B 0,C 180,E1 -15760.419,E2 -15760.419} C_VEL
LIN {X 0,Y 310.718,Z 524.837,A -85,B 0,C 180,E1 -15761.744,E2 -15761.744} C_VEL
LIN {X 0,Y 310.627,Z 526.385,A -85,B 0,C 180,E1 -15763.374,E2 -15763.374} C_VEL
LIN {X 0,Y 310.544,Z 527.453,A -85,B 0,C 180,E1 -15765.756,E2 -15765.756} C_VEL
LIN {X 0,Y 310.761,Z 527.183,A -85,B 0,C 180,E1 -15768.223,E2 -15768.223} C_VEL
LIN {X 0,Y 310.988,Z 526.264,A -85,B 0,C 180,E1 -15769.813,E2 -15769.813} C_VEL
LIN {X 0,Y 311.63,Z 523.474,A -85,B 0,C 180,E1 -15772.385,E2 -15772.385} C_VEL
LIN {X 0,Y 312.429,Z 519.761,A -85,B 0,C 180,E1 -15774.589,E2 -15774.589} C_VEL
LIN {X 0,Y 313.431,Z 515.041,A -85,B 0,C 180,E1 -15776.642,E2 -15776.642} C_VEL
LIN {X 0,Y 314.741,Z 508.922,A -85,B 0,C 180,E1 -15778.688,E2 -15778.688} C_VEL
LIN {X 0,Y 316.386,Z 501.187,A -85,B 0,C 180,E1 -15780.722,E2 -15780.722} C_VEL
LIN {X 0,Y 317.957,Z 493.543,A -85,B 0,C 180,E1 -15782.336,E2 -15782.336} C_VEL
LIN {X 0,Y 319.566,Z 484.43,A -85,B 0,C 180,E1 -15783.919,E2 -15783.919} C_VEL
LIN {X 0,Y 321.496,Z 473.574,A -85,B 0,C 180,E1 -15785.398,E2 -15785.398} C_VEL
LIN {X 0,Y 323.23,Z 461.562,A -85,B 0,C 180,E1 -15786.694,E2 -15786.694} C_VEL
LIN {X 0,Y 324.607,Z 449.2,A -85,B 0,C 180,E1 -15787.705,E2 -15787.705} C_VEL
LIN {X 0,Y 325.809,Z 436.097,A -85,B 0,C 180,E1 -15788.473,E2 -15788.473} C_VEL
LIN {X 0,Y 326.52,Z 423.737,A -85,B 0,C 180,E1 -15788.959,E2 -15788.959} C_VEL
LIN {X 0,Y 328.725,Z 349.266,A -85,B 0,C 180,E1 -15790.633,E2 -15790.633} C_VEL
LIN {X 0,Y 324.397,Z 338.566,A -85,B 0,C 180,E1 -15791.358,E2 -15791.358} C_VEL
LIN {X 0,Y 317.444,Z 324.074,A -85,B 0,C 180,E1 -15792.506,E2 -15792.506} C_VEL
LIN {X 0,Y 314.036,Z 317.362,A -85,B 0,C 180,E1 -15793.084,E2 -15793.084} C_VEL
LIN {X 0,Y 311.521,Z 316.292,A -85,B 0,C 180,E1 -15793.67,E2 -15793.67} C_VEL
LIN {X 0,Y 308.075,Z 314.679,A -85,B 0,C 180,E1 -15794.737,E2 -15794.737} C_VEL
LIN {X 0,Y 305.989,Z 313.1,A -85,B 0,C 180,E1 -15795.749,E2 -15795.749} C_VEL
LIN {X 0,Y 305.404,Z 312.433,A -85,B 0,C 180,E1 -15796.566,E2 -15796.566} C_VEL
